	// Sensors - Waster Water Sump
	{attribute 'OPC.UA.DA' := '1'}
  	{attribute 'OPC.UA.DA.StructuredType' := '1'}
	fbSensor_WWS_LSLL : FB_Sensor_SICKLevelSwitch_GRF18S(SensorID:= 'SU3-LSLL' , SensorDescr:= 'Waste Water Sump Level Switch - LOW LOW', SensorType:= E_SensorType.Analogue);
	{attribute 'OPC.UA.DA' := '1'}
  	{attribute 'OPC.UA.DA.StructuredType' := '1'}
	fbSensor_WWS_LSL : FB_Sensor_SICKLevelSwitch_GRF18S(SensorID:= 'SU3-LSL' , SensorDescr:= 'Waste Water Sump Level Switch - LOW', SensorType:= E_SensorType.Analogue);
	{attribute 'OPC.UA.DA' := '1'}
  	{attribute 'OPC.UA.DA.StructuredType' := '1'}
	fbSensor_WWS_LSH : FB_Sensor_SICKLevelSwitch_GRF18S(SensorID:= 'SU3-LSH' , SensorDescr:= 'Waste Water Sump Level Switch - HIGH', SensorType:= E_SensorType.Analogue);
	
	
	// Sensors - Waster Water Tank
	{attribute 'OPC.UA.DA' := '1'}
  	{attribute 'OPC.UA.DA.StructuredType' := '1'}
	fbSensor_WWT_LIT1 : FB_Sensor_4_20mA_Generic(SensorID:= 'TK1-LIT1', SensorDescr:= 'Waste Water Tank Level Transmitter 1' , SensorType:= E_SensorType.Analogue);
	{attribute 'OPC.UA.DA' := '1'}
  	{attribute 'OPC.UA.DA.StructuredType' := '1'} 
	fbSensor_WWT_LIT2 : FB_Sensor_4_20mA_Generic(SensorID:= 'TK1-LIT1', SensorDescr:= 'Waste Water Tank Level Transmitter 2' , SensorType:= E_SensorType.Analogue);
	{attribute 'OPC.UA.DA' := '1'}
  	{attribute 'OPC.UA.DA.StructuredType' := '1'}
 	fbSensor_WWT_LIT : FB_DualRedundantSensor(SensorID:= 'TK1-LIT', SensorDescr:= 'Waste Water Tank Level', SensorType:= E_SensorType.Analogue);
	
	// Actuated Valves 
	{attribute 'OPC.UA.DA' := '1'}
  	{attribute 'OPC.UA.DA.StructuredType' := '1'}
	fbValve_TownWaterSupply: FB_Valve_ONOFF_woMonitoring(ValveID:= 'TK1-V2', ValveDescr:= 'Town Water Supply Valve');
	{attribute 'OPC.UA.DA' := '1'}
  	{attribute 'OPC.UA.DA.StructuredType' := '1'}
	fbValve_DosingSupply: FB_Valve_ONOFF_woMonitoring(ValveID:= 'PU1-V1', ValveDescr:= 'Dosing Circuit Supply Valve');
	{attribute 'OPC.UA.DA' := '1'}
  	{attribute 'OPC.UA.DA.StructuredType' := '1'}
	fbValve_DM1Supply: FB_Valve_ONOFF_woMonitoring(ValveID:= 'PU1-V2', ValveDescr:= 'Dosing Machine 1 Supply Valve' );
	{attribute 'OPC.UA.DA' := '1'}
  	{attribute 'OPC.UA.DA.StructuredType' := '1'} 
	fbValve_DM2Supply: FB_Valve_ONOFF_woMonitoring(ValveID:= 'PU1-V3', ValveDescr:= 'Dosing Machine 2 Supply Valve' );
	{attribute 'OPC.UA.DA' := '1'}
  	{attribute 'OPC.UA.DA.StructuredType' := '1'}
	fbValve_SeedStackSupply: FB_Valve_ONOFF_woMonitoring(ValveID:= 'PU1-V4', ValveDescr:= 'Seedling Stack Supply Valve' );
	{attribute 'OPC.UA.DA' := '1'}
  	{attribute 'OPC.UA.DA.StructuredType' := '1'}
	fbValve_SDRSoakSupply: FB_Valve_ONOFF_woMonitoring(ValveID:= 'PU1-V5', ValveDescr:= 'SDR Soak Supply Valve' );
	{attribute 'OPC.UA.DA' := '1'}
  	{attribute 'OPC.UA.DA.StructuredType' := '1'} 
	fbValve_WashSupply: FB_Valve_ONOFF_woMonitoring(ValveID:= 'PU1-V6', ValveDescr:= 'Pressure Wash Pumps Supply' );
	{attribute 'OPC.UA.DA' := '1'}
  	{attribute 'OPC.UA.DA.StructuredType' := '1'}
	fbValve_FogMistSupply: FB_Valve_ONOFF_woMonitoring(ValveID:= 'PU1-V7', ValveDescr:= 'Fog and Misting Pumps Supply' ); 

	// Tanks and Sumps
	{attribute 'OPC.UA.DA' := '1'}
  	{attribute 'OPC.UA.DA.StructuredType' := '1'}
	fbTank_CWTA: FB_Tank(TankID:= 'TK1A', TankDescr:= 'Clean Water Tank A');
	{attribute 'OPC.UA.DA' := '1'}
  	{attribute 'OPC.UA.DA.StructuredType' := '1'}
	fbTank_CWTB: FB_Tank(TankID:= 'TK1B', TankDescr:= 'Clean Water Tank B');
	{attribute 'OPC.UA.DA' := '1'}
  	{attribute 'OPC.UA.DA.StructuredType' := '1'}
	fbTank_WWT: FB_Tank(TankID:= 'TK2', TankDescr:= 'Waste Water Tank');
	{attribute 'OPC.UA.DA' := '1'}
  	{attribute 'OPC.UA.DA.StructuredType' := '1'}
	fbSump_WWS: FB_Tank(TankID:= 'TK3', TankDescr:= 'Waste Water Sump');
	
	
	// Control Loops
{attribute 'OPC.UA.DA' := '0'}
	fbControlLoop_Dosing: FB_ControlLoop_pH(
								DosingPump_phUp := fbDosingPump_phUp, 
								DosingPump_phDOwn := fbDosingPump_phDown, 
								Sensor_PH := fbSensor_PH, 
								Sensor_TEMP := fbSensor_TMP);
	
	
	// Package all components into structure to pass to sub-FBs 
	// This ST is populated by calling the populateComponents method
	{attribute 'OPC.UA.DA' := '0'} 
	stAllComponents: ST_WTRComponents;
	
	
	// Interlocks
	{attribute 'OPC.UA.DA' := '1'}
  	{attribute 'OPC.UA.DA.StructuredType' := '1'}
	fbInterlocks: FB_InterlockManager;
	
	{attribute 'OPC.UA.DA' := '1'}
	bInCalibration: BOOL := FALSE;
	
	// Sequence Manager & Sequences
	{attribute 'OPC.UA.DA' := '0'}
	fbSeqWTRMain: FB_SequenceWTR_Main;
	{attribute 'OPC.UA.DA' := '0'}
	fbSeqWTRMCalibrate: FB_SequenceWTR_Calibrate;
	{attribute 'OPC.UA.DA' := '0'}
	aSeqs: ARRAY[1..5] OF FB_SequenceBase;
	
END_VAR

IF GVL.bAutoUpdateDeviceState THEN
	simulation();       //  <<<----------------- FOR TESTING ONLY, delete this when not being used (it changes devices statet to the target state automatically)
END_IF

IF bIsFirstRun  THEN
	devices_init();	
	sequence_init();
	bIsFirstRun := FALSE;
END_IF


scanOPCInputs();
fbSequenceManager(aSequences := aSeqs, fbCurrentSequence := aSeqs[1]);
fbControlLoop_Dosing();

IF GVL.bEnableInterlocks_DM THEN
	interlocks();
END_IF

devices_update();

METHOD checkWaterQuality : BOOL
VAR_INPUT
END_VAR
(*

checkWaterQuality := TRUE;

IF fbSensor_PH.getValue() > stInputs.PH_HIGH_Limit OR 
	fbSensor_PH.getValue() < stInputs.PH_LOW_Limit THEN
	
	checkWaterQuality := FALSE;
	// Raise an event to alert that PH is out of range
END_IF

IF fbSensor_TMP.getValue() > stInputs.Temp_HIGH_Limit OR
	fbSensor_TMP.getValue() < stInputs.Temp_LOW_Limit THEN
	
	checkWaterQuality := FALSE;
	// Raise an event to alert that temp is out of range
END_IF

*)
END_METHOD

METHOD devices_init : BOOL
VAR
	VarInfo : __SYSTEM.VAR_INFO;
END_VAR
fbSump_WWS.fbSensor_LL := fbSensor_WWS_LSLL;
fbSump_WWS.fbSensor_L := fbSensor_WWS_LSL;
fbSump_WWS.fbSensor_H := fbSensor_WWS_LSH;
fbSump_WWS.fbSensor_HH := fbSensor_WWT_LIT;
fbSump_WWS.fbSensor_LIT := fbSensor_WWT_LIT;

fbTank_CWTA.fbSensor_LL := fbSensor_CWT_A_LSLL;
fbTank_CWTA.fbSensor_L := fbSensor_CWT_A_LSL;
fbTank_CWTA.fbSensor_H := fbSensor_CWT_A_LSH;
fbTank_CWTA.fbSensor_HH := fbSensor_CWT_A_LSHH;
fbTank_CWTA.fbSensor_LIT := fbSensor_CWT_A_LSHH;

fbTank_CWTB.fbSensor_LL := fbSensor_CWT_A_LSLL;
fbTank_CWTB.fbSensor_L := fbSensor_CWT_A_LSL;
fbTank_CWTB.fbSensor_H := fbSensor_CWT_A_LSH;
fbTank_CWTB.fbSensor_HH := fbSensor_CWT_A_LSHH;
fbTank_CWTB.fbSensor_LIT := fbSensor_CWT_A_LSHH;

fbTank_WWT.fbSensor_LL := fbSensor_CWT_A_LSLL;
fbTank_WWT.fbSensor_L := fbSensor_CWT_A_LSL;
fbTank_WWT.fbSensor_H := fbSensor_CWT_A_LSH;
fbTank_WWT.fbSensor_HH := fbSensor_CWT_A_LSHH;
fbTank_WWT.fbSensor_LIT := fbSensor_CWT_A_LSHH;




VarInfo := __VARINFO(fbDosingPump_phDown);
fbDosingPump_phDown.setVarID(VarID := VarInfo.Symbol);
VarInfo := __VARINFO(fbDosingPump_phUp);
fbDosingPump_phUp.setVarID(VarID := VarInfo.Symbol);
VarInfo := __VARINFO(fbDrumFilter_WasteWaterSump);
fbDrumFilter_WasteWaterSump.setVarID(VarID := VarInfo.Symbol);
VarInfo := __VARINFO(fbPump_CleanWaterPumpA);
fbPump_CleanWaterPumpA.setVarID(VarID := VarInfo.Symbol);
VarInfo := __VARINFO(fbPump_CleanWaterPumpB);
fbPump_CleanWaterPumpB.setVarID(VarID := VarInfo.Symbol);
VarInfo := __VARINFO(fbPump_WasteWaterSumpPumpA );
fbPump_WasteWaterSumpPumpA .setVarID(VarID := VarInfo.Symbol);
VarInfo := __VARINFO(fbPump_WasteWaterSumpPumpB );
fbPump_WasteWaterSumpPumpB .setVarID(VarID := VarInfo.Symbol);
VarInfo := __VARINFO(fbSensor_CWT_A_LIT );
fbSensor_CWT_A_LIT .setVarID(VarID := VarInfo.Symbol);
VarInfo := __VARINFO(fbSensor_CWT_A_LIT1 );
fbSensor_CWT_A_LIT1 .setVarID(VarID := VarInfo.Symbol);
VarInfo := __VARINFO(fbSensor_CWT_A_LIT2 );
fbSensor_CWT_A_LIT2 .setVarID(VarID := VarInfo.Symbol);
VarInfo := __VARINFO(fbSensor_CWT_A_LSH );
fbSensor_CWT_A_LSH .setVarID(VarID := VarInfo.Symbol);
VarInfo := __VARINFO(fbSensor_CWT_A_LSHH );
fbSensor_CWT_A_LSHH .setVarID(VarID := VarInfo.Symbol);
VarInfo := __VARINFO(fbSensor_CWT_A_LSL );
fbSensor_CWT_A_LSL .setVarID(VarID := VarInfo.Symbol);
VarInfo := __VARINFO(fbSensor_CWT_A_LSLL );
fbSensor_CWT_A_LSLL .setVarID(VarID := VarInfo.Symbol);
VarInfo := __VARINFO(fbSensor_CWT_B_LIT );
fbSensor_CWT_B_LIT .setVarID(VarID := VarInfo.Symbol);
VarInfo := __VARINFO(fbSensor_CWT_B_LIT1 );
fbSensor_CWT_B_LIT1 .setVarID(VarID := VarInfo.Symbol);
VarInfo := __VARINFO(fbSensor_CWT_B_LIT2 );
fbSensor_CWT_B_LIT2 .setVarID(VarID := VarInfo.Symbol);
VarInfo := __VARINFO(fbSensor_CWT_B_LSH );
fbSensor_CWT_B_LSH .setVarID(VarID := VarInfo.Symbol);
VarInfo := __VARINFO(fbSensor_CWT_B_LSHH );
fbSensor_CWT_B_LSHH .setVarID(VarID := VarInfo.Symbol);
VarInfo := __VARINFO(fbSensor_CWT_B_LSL );
fbSensor_CWT_B_LSL .setVarID(VarID := VarInfo.Symbol);
VarInfo := __VARINFO(fbSensor_CWT_B_LSLL );
fbSensor_CWT_B_LSLL .setVarID(VarID := VarInfo.Symbol);
VarInfo := __VARINFO(fbSensor_PH);
fbSensor_PH.setVarID(VarID := VarInfo.Symbol);
VarInfo := __VARINFO(fbSensor_PH1);
fbSensor_PH1.setVarID(VarID := VarInfo.Symbol);
VarInfo := __VARINFO(fbSensor_PH2);
fbSensor_PH2.setVarID(VarID := VarInfo.Symbol);
VarInfo := __VARINFO(fbSensor_TMP);
fbSensor_TMP.setVarID(VarID := VarInfo.Symbol);
VarInfo := __VARINFO(fbSensor_TMP1);
fbSensor_TMP1.setVarID(VarID := VarInfo.Symbol);
VarInfo := __VARINFO(fbSensor_TMP2);
fbSensor_TMP2.setVarID(VarID := VarInfo.Symbol);
VarInfo := __VARINFO(fbSensor_WWS_LSH );
fbSensor_WWS_LSH .setVarID(VarID := VarInfo.Symbol);
VarInfo := __VARINFO(fbSensor_WWS_LSL );
fbSensor_WWS_LSL .setVarID(VarID := VarInfo.Symbol);
VarInfo := __VARINFO(fbSensor_WWS_LSLL );
fbSensor_WWS_LSLL .setVarID(VarID := VarInfo.Symbol);
VarInfo := __VARINFO(fbSensor_WWT_LIT );
fbSensor_WWT_LIT .setVarID(VarID := VarInfo.Symbol);
VarInfo := __VARINFO(fbSensor_WWT_LIT1 );
fbSensor_WWT_LIT1 .setVarID(VarID := VarInfo.Symbol);
VarInfo := __VARINFO(fbSensor_WWT_LIT2 );
fbSensor_WWT_LIT2 .setVarID(VarID := VarInfo.Symbol);
VarInfo := __VARINFO(fbSump_WWS);
fbSump_WWS.setVarID(VarID := VarInfo.Symbol);
VarInfo := __VARINFO(fbTank_CWTA);
fbTank_CWTA.setVarID(VarID := VarInfo.Symbol);
VarInfo := __VARINFO(fbTank_CWTB);
fbTank_CWTB.setVarID(VarID := VarInfo.Symbol);
VarInfo := __VARINFO(fbTank_WWT);
fbTank_WWT.setVarID(VarID := VarInfo.Symbol);
VarInfo := __VARINFO(fbUnit_OzoneGenerator);
fbUnit_OzoneGenerator.setVarID(VarID := VarInfo.Symbol);
VarInfo := __VARINFO(fbUnit_RO_EDI);
fbUnit_RO_EDI.setVarID(VarID := VarInfo.Symbol);
VarInfo := __VARINFO(fbValve_DM1Supply);
fbValve_DM1Supply.setVarID(VarID := VarInfo.Symbol);
VarInfo := __VARINFO(fbValve_DM2Supply);
fbValve_DM2Supply.setVarID(VarID := VarInfo.Symbol);
VarInfo := __VARINFO(fbValve_DosingSupply);
fbValve_DosingSupply.setVarID(VarID := VarInfo.Symbol);
VarInfo := __VARINFO(fbValve_FogMistSupply);
fbValve_FogMistSupply.setVarID(VarID := VarInfo.Symbol);
VarInfo := __VARINFO(fbValve_SDRSoakSupply);
fbValve_SDRSoakSupply.setVarID(VarID := VarInfo.Symbol);
VarInfo := __VARINFO(fbValve_SeedStackSupply);
fbValve_SeedStackSupply.setVarID(VarID := VarInfo.Symbol);
VarInfo := __VARINFO(fbValve_TownWaterSupply);
fbValve_TownWaterSupply.setVarID(VarID := VarInfo.Symbol);
VarInfo := __VARINFO(fbValve_WashSupply);
fbValve_WashSupply.setVarID(VarID := VarInfo.Symbol);




stAllComponents.fbDosingPump_phUp :=  ADR( fbDosingPump_phUp);
stAllComponents.fbDosingPump_phDown :=  ADR( fbDosingPump_phDown);
stAllComponents.fbPump_CleanWaterPumpA :=  ADR( fbPump_CleanWaterPumpA);
stAllComponents.fbPump_CleanWaterPumpB :=  ADR( fbPump_CleanWaterPumpB);
stAllComponents.fbPump_WasteWaterSumpPumpA :=  ADR( fbPump_WasteWaterSumpPumpA);
stAllComponents.fbPump_WasteWaterSumpPumpB :=  ADR( fbPump_WasteWaterSumpPumpB);
stAllComponents.fbUnit_OzoneGenerator :=  ADR( fbUnit_OzoneGenerator);
stAllComponents.fbUnit_RO_EDI := ADR( fbUnit_RO_EDI);
stAllComponents.fbDrumFilter_WasteWaterSump :=  ADR( fbDrumFilter_WasteWaterSump);
stAllComponents.fbSensor_PH1 :=  ADR( fbSensor_PH1);
stAllComponents.fbSensor_PH2 :=  ADR( fbSensor_PH2);
stAllComponents.fbSensor_PH :=  ADR( fbSensor_PH);
stAllComponents.fbSensor_TMP1 :=  ADR( fbSensor_TMP1);
stAllComponents.fbSensor_TMP2 :=  ADR( fbSensor_TMP2);
stAllComponents.fbSensor_TMP :=  ADR( fbSensor_TMP);
stAllComponents.fbSensor_CWT_A_LIT1 :=  ADR( fbSensor_CWT_A_LIT1);
stAllComponents.fbSensor_CWT_A_LIT2 :=  ADR( fbSensor_CWT_A_LIT2);
stAllComponents.fbSensor_CWT_A_LIT :=  ADR( fbSensor_CWT_A_LIT);
stAllComponents.fbSensor_CWT_A_LSLL :=  ADR( fbSensor_CWT_A_LSLL);
stAllComponents.fbSensor_CWT_A_LSL :=  ADR( fbSensor_CWT_A_LSL);
stAllComponents.fbSensor_CWT_A_LSH :=  ADR( fbSensor_CWT_A_LSH);
stAllComponents.fbSensor_CWT_A_LSHH :=  ADR( fbSensor_CWT_A_LSHH);
stAllComponents.fbSensor_CWT_B_LIT1 :=  ADR( fbSensor_CWT_B_LIT1);
stAllComponents.fbSensor_CWT_B_LIT2 :=  ADR( fbSensor_CWT_B_LIT2);
stAllComponents.fbSensor_CWT_B_LIT :=  ADR( fbSensor_CWT_B_LIT);
stAllComponents.fbSensor_CWT_B_LSLL :=  ADR( fbSensor_CWT_B_LSLL);
stAllComponents.fbSensor_CWT_B_LSL :=  ADR( fbSensor_CWT_B_LSL);
stAllComponents.fbSensor_CWT_B_LSH :=  ADR( fbSensor_CWT_B_LSH);
stAllComponents.fbSensor_CWT_B_LSHH :=  ADR( fbSensor_CWT_B_LSHH);
stAllComponents.fbSensor_WWS_LSLL :=  ADR( fbSensor_WWS_LSLL);
stAllComponents.fbSensor_WWS_LSL :=  ADR( fbSensor_WWS_LSL);
stAllComponents.fbSensor_WWS_LSH :=  ADR( fbSensor_WWS_LSH);
stAllComponents.fbSensor_WWT_LIT1 :=  ADR( fbSensor_WWT_LIT1);
stAllComponents.fbSensor_WWT_LIT2 :=  ADR( fbSensor_WWT_LIT2);
stAllComponents.fbSensor_WWT_LIT :=  ADR( fbSensor_WWT_LIT);
stAllComponents.fbValve_TownWaterSupply :=  ADR( fbValve_TownWaterSupply);
stAllComponents.fbValve_DosingSupply :=  ADR( fbValve_DosingSupply);
stAllComponents.fbValve_DM1Supply :=  ADR( fbValve_DM1Supply);
stAllComponents.fbValve_DM2Supply :=  ADR( fbValve_DM2Supply);
stAllComponents.fbValve_SeedStackSupply :=  ADR( fbValve_SeedStackSupply);
stAllComponents.fbValve_SDRSoakSupply :=  ADR( fbValve_SDRSoakSupply);
stAllComponents.fbValve_WashSupply :=  ADR( fbValve_WashSupply);
stAllComponents.fbValve_FogMistSupply :=  ADR( fbValve_FogMistSupply);
stAllComponents.fbTank_CWTA :=  ADR( fbTank_CWTA);
stAllComponents.fbTank_CWTB :=  ADR( fbTank_CWTB);
stAllComponents.fbTank_WWT :=  ADR( fbTank_WWT);
stAllComponents.fbSump_WWS :=  ADR( fbSump_WWS);


aAllComponents[1]  :=  ADR(fbPump_CleanWaterPumpA );
aAllComponents[2]  :=  ADR(fbPump_CleanWaterPumpB );
aAllComponents[3]  :=  ADR(fbPump_WasteWaterSumpPumpA  );
aAllComponents[4]  :=  ADR(fbPump_WasteWaterSumpPumpB  );
aAllComponents[5]  :=  ADR(fbUnit_OzoneGenerator );
aAllComponents[6]  :=  ADR(fbDrumFilter_WasteWaterSump );
aAllComponents[7]  :=  ADR(fbUnit_RO_EDI );
aAllComponents[8]  :=  ADR(fbSensor_PH1 );
aAllComponents[9]  :=  ADR(fbSensor_PH2 );
aAllComponents[10]  :=  ADR(fbSensor_PH );
aAllComponents[11]  :=  ADR(fbSensor_TMP1 );
aAllComponents[12]  :=  ADR(fbSensor_TMP2 );
aAllComponents[13]  :=  ADR(fbSensor_TMP );
aAllComponents[14]  :=  ADR(fbSensor_CWT_A_LIT1  );
aAllComponents[15]  :=  ADR(fbSensor_CWT_A_LIT2  );
aAllComponents[16]  :=  ADR(fbSensor_CWT_A_LIT  );
aAllComponents[17]  :=  ADR(fbSensor_CWT_A_LSLL  );
aAllComponents[18]  :=  ADR(fbSensor_CWT_A_LSL  );
aAllComponents[19]  :=  ADR(fbSensor_CWT_A_LSH  );
aAllComponents[20]  :=  ADR(fbSensor_CWT_A_LSHH  );
aAllComponents[21]  :=  ADR(fbSensor_CWT_B_LIT1  );
aAllComponents[22]  :=  ADR(fbSensor_CWT_B_LIT2  );
aAllComponents[23]  :=  ADR(fbSensor_CWT_B_LIT  );
aAllComponents[24]  :=  ADR(fbSensor_CWT_B_LSLL  );
aAllComponents[25]  :=  ADR(fbSensor_CWT_B_LSL  );
aAllComponents[26]  :=  ADR(fbSensor_CWT_B_LSH  );
aAllComponents[27]  :=  ADR(fbSensor_CWT_B_LSHH  );
aAllComponents[28]  :=  ADR(fbSensor_WWS_LSLL  );
aAllComponents[29]  :=  ADR(fbSensor_WWS_LSL  );
aAllComponents[30]  :=  ADR(fbSensor_WWS_LSH  );
aAllComponents[31]  :=  ADR(fbSensor_WWT_LIT1  );
aAllComponents[32]  :=  ADR(fbSensor_WWT_LIT2  );
aAllComponents[33]  :=  ADR(fbSensor_WWT_LIT  );
aAllComponents[34]  :=  ADR(fbValve_TownWaterSupply );
aAllComponents[35]  :=  ADR(fbValve_DosingSupply );
aAllComponents[36]  :=  ADR(fbValve_DM1Supply );
aAllComponents[37]  :=  ADR(fbValve_DM2Supply );
aAllComponents[38]  :=  ADR(fbValve_SeedStackSupply );
aAllComponents[39]  :=  ADR(fbValve_SDRSoakSupply );
aAllComponents[40]  :=  ADR(fbValve_WashSupply );
aAllComponents[41]  :=  ADR(fbValve_FogMistSupply );
aAllComponents[42]  :=  ADR(fbTank_CWTA );
aAllComponents[43]  :=  ADR(fbTank_CWTB );
aAllComponents[44]  :=  ADR(fbTank_WWT );
aAllComponents[45]  :=  ADR(fbSump_WWS );

nQtyComponents := 45;
devices_disable_All();
END_METHOD

METHOD devices_update : BOOL
VAR_INPUT
END_VAR
fbModbusMaster();

fbDosingPump_phUp(fbModbusMaster := fbModbusMaster);
fbDosingPump_phDown(fbModbusMaster := fbModbusMaster);
fbPump_CleanWaterPumpA(fbModbusMaster := fbModbusMaster);	 
fbPump_CleanWaterPumpB(fbModbusMaster := fbModbusMaster); 
fbPump_WasteWaterSumpPumpA();
fbPump_WasteWaterSumpPumpB();
fbUnit_OzoneGenerator();
fbDrumFilter_WasteWaterSump();
fbSensor_PH1();
fbSensor_PH2();
fbSensor_PH();
fbSensor_TMP1();
fbSensor_TMP2();
fbSensor_TMP();
fbSensor_CWT_A_LIT1(); 
fbSensor_CWT_A_LIT2();
fbSensor_CWT_A_LIT();
fbSensor_CWT_A_LSLL();
fbSensor_CWT_A_LSL();
fbSensor_CWT_A_LSH();
fbSensor_CWT_A_LSHH();
fbSensor_CWT_B_LIT1(); 
fbSensor_CWT_B_LIT2();
fbSensor_CWT_B_LIT();
fbSensor_CWT_B_LSLL();
fbSensor_CWT_B_LSL();
fbSensor_CWT_B_LSH();
fbSensor_CWT_B_LSHH();
fbSensor_WWS_LSLL();
fbSensor_WWS_LSL();
fbSensor_WWS_LSH();
fbSensor_WWT_LIT1(); 
fbSensor_WWT_LIT2();
fbSensor_WWT_LIT();
fbValve_TownWaterSupply();
fbValve_DosingSupply();
fbValve_DM1Supply(); 
fbValve_DM2Supply();
fbValve_SeedStackSupply();
fbValve_SDRSoakSupply(); 
fbValve_WashSupply();
fbValve_FogMistSupply(); 
fbTank_CWTA();
fbTank_CWTB();		
fbTank_WWT();	
fbSump_WWS();
END_METHOD

METHOD FB_init : BOOL
VAR_INPUT
	bInitRetains : BOOL; // if TRUE, the retain variables are initialized (warm start / cold start)
	bInCopyCode : BOOL;  // if TRUE, the instance afterwards gets moved into the copy code (online change)


END_VAR
END_METHOD

METHOD interlocks : BOOL
VAR_INPUT
END_VAR


fbInterlocks.init();



// Dosing Pump - PH Up Interlocks

							
fbInterlocks.update(
							Description:= 'PH Down Dosing Pump - RUNNING',
							InterlockType:= E_InterlockType.RunInterlock, 
							Subject_Device:= ADR(fbDosingPump_phUp), 
							Subject_State:= E_DeviceState.IDLE, 
							Signal:= fbDosingPump_phDown.getState() = E_DeviceState.RUNNING, 
							HoldSequence:=	TRUE );
					
							
fbInterlocks.update(
							Description:= 'Dosing Line Pressure - OUT OF RANGE',		
							InterlockType:= E_InterlockType.StartPermissive, 
							Subject_Device:= ADR(fbDosingPump_phUp), 
							Subject_State:= E_DeviceState.IDLE, 
							Signal:= fbSensor_DosingPIT1.getState() = E_DeviceState.OUT_OF_RANGE, 
							HoldSequence:=	FALSE );	
							
// Dosing Pump - PH Down Interlocks


fbInterlocks.update(
							Description:= 'PH Up Dosing Pump - RUNNING',		
							InterlockType:= E_InterlockType.RunInterlock, 
							Subject_Device:= ADR(fbDosingPump_phDown), 
							Subject_State:= E_DeviceState.IDLE, 
							Signal:= fbDosingPump_phUp.getState() = E_DeviceState.RUNNING, 
							HoldSequence:=	TRUE );
							
fbInterlocks.update(
							Description:= 'Dosing Line Pressure - OUT OF RANGE',		
							InterlockType:= E_InterlockType.RunInterlock, 
							Subject_Device:= ADR(fbDosingPump_phDown), 
							Subject_State:= E_DeviceState.IDLE, 
							Signal:= fbSensor_DosingPIT1.getState() = E_DeviceState.OUT_OF_RANGE, 
							HoldSequence:=	FALSE );

							
// Clean Water Pump A - Interlocks	


fbInterlocks.update(
							Description:= 'Clean Water Pump B - RUNNING', 
							InterlockType:= E_InterlockType.RunInterlock, 
							Subject_Device:= ADR(fbPump_CleanWaterPumpA), 
							Subject_State:= E_DeviceState.IDLE, 
							Signal:= fbPump_CleanWaterPumpB.getState() = E_DeviceState.RUNNING, 
							HoldSequence:= TRUE);

fbInterlocks.update(
							Description:= 'Pressure Transmitter - OUT OF RANGE', 
							InterlockType:= E_InterlockType.RunInterlock, 
							Subject_Device:= ADR(fbPump_CleanWaterPumpA), 
							Subject_State:= E_DeviceState.IDLE, 
							Signal:= fbSensor_MainPumpPIT1.getState() = E_DeviceState.OUT_OF_RANGE, 
							HoldSequence:= TRUE);

fbInterlocks.update(
							Description:= 'Clean Water Tank (A) - LOW LOW Level', 
							InterlockType:= E_InterlockType.RunInterlock, 
							Subject_Device:= ADR(fbPump_CleanWaterPumpA), 
							Subject_State:= E_DeviceState.IDLE, 
							Signal:= fbTank_CWTA.getState() = E_DeviceState.LOW_LOW, 
							HoldSequence:= TRUE);

fbInterlocks.update(
							Description:= 'Clean Water Tank (B) - LOW LOW Level', 
							InterlockType:= E_InterlockType.RunInterlock, 
							Subject_Device:= ADR(fbPump_CleanWaterPumpA), 
							Subject_State:= E_DeviceState.IDLE, 
							Signal:= fbTank_CWTB.getState() = E_DeviceState.LOW_LOW, 
							HoldSequence:= TRUE);
							
fbInterlocks.update(
							Description:= 'Valve Combination - DM1, DM2, Recirc, Fog, SDR, Seedstack and Wash - CLOSED', 
							InterlockType:= E_InterlockType.RunInterlock, 
							Subject_Device:= ADR(fbPump_CleanWaterPumpA), 
							Subject_State:= E_DeviceState.IDLE, 
							Signal:= fbTank_CWTB.getState() = E_DeviceState.LOW_LOW, 
							HoldSequence:= TRUE);

// Clean Water Pump B - Interlocks	


fbInterlocks.update(
							Description:= 'Clean Water Pump A - RUNNING', 
							InterlockType:= E_InterlockType.RunInterlock, 
							Subject_Device:= ADR(fbPump_CleanWaterPumpB), 
							Subject_State:= E_DeviceState.IDLE, 
							Signal:= fbPump_CleanWaterPumpA.getState() = E_DeviceState.RUNNING, 
							HoldSequence:= TRUE);

fbInterlocks.update(
							Description:= 'Pressure Transmitter - OUT OF RANGE', 
							InterlockType:= E_InterlockType.RunInterlock, 
							Subject_Device:= ADR(fbPump_CleanWaterPumpB), 
							Subject_State:= E_DeviceState.IDLE, 
							Signal:= fbSensor_MainPumpPIT1.getState() = E_DeviceState.OUT_OF_RANGE, 
							HoldSequence:= TRUE);

fbInterlocks.update(
							Description:= 'Clean Water Tank (A) - LOW LOW Level', 
							InterlockType:= E_InterlockType.RunInterlock, 
							Subject_Device:= ADR(fbPump_CleanWaterPumpB), 
							Subject_State:= E_DeviceState.IDLE, 
							Signal:= fbTank_CWTA.getState() = E_DeviceState.LOW_LOW, 
							HoldSequence:= TRUE);

fbInterlocks.update(
							Description:= 'Clean Water Tank (B) - LOW LOW Level', 
							InterlockType:= E_InterlockType.RunInterlock, 
							Subject_Device:= ADR(fbPump_CleanWaterPumpB), 
							Subject_State:= E_DeviceState.IDLE, 
							Signal:= fbTank_CWTB.getState() = E_DeviceState.LOW_LOW, 
							HoldSequence:= TRUE);
							
fbInterlocks.update(
							Description:= 'Valve Combination - DM1, DM2, Recirc, Fog, SDR, Seedstack and Wash - CLOSED', 
							InterlockType:= E_InterlockType.RunInterlock, 
							Subject_Device:= ADR(fbPump_CleanWaterPumpB), 
							Subject_State:= E_DeviceState.IDLE, 
							Signal:= fbTank_CWTB.getState() = E_DeviceState.LOW_LOW, 
							HoldSequence:= TRUE);

// Waste Water Sump (WWS) Pump A							
							
fbInterlocks.update(
							Description:= 'Waste Water Sump Pump B - RUNNING', 
							InterlockType:= E_InterlockType.RunInterlock, 
							Subject_Device:= ADR(fbPump_WasteWaterSumpPumpA), 
							Subject_State:= E_DeviceState.IDLE, 
							Signal:= fbPump_WasteWaterSumpPumpB.getState() = E_DeviceState.RUNNING, 
							HoldSequence:= TRUE);
							
fbInterlocks.update(
							Description:= 'Waste Water Sump - LOW LOW Level', 
							InterlockType:= E_InterlockType.RunInterlock, 
							Subject_Device:= ADR(fbPump_WasteWaterSumpPumpA), 
							Subject_State:= E_DeviceState.IDLE, 
							Signal:= fbSump_WWS.getState() = E_DeviceState.LOW_LOW, 
							HoldSequence:= TRUE);		


// Waste Water Sump (WWS) Pump B							
							
fbInterlocks.update(
							Description:= 'Waste Water Sump Pump A - RUNNING', 
							InterlockType:= E_InterlockType.RunInterlock, 
							Subject_Device:= ADR(fbPump_WasteWaterSumpPumpB), 
							Subject_State:= E_DeviceState.IDLE, 
							Signal:= fbPump_WasteWaterSumpPumpA.getState() = E_DeviceState.RUNNING, 
							HoldSequence:= TRUE);
							
fbInterlocks.update(
							Description:= 'Waste Water Sump - LOW LOW Level', 
							InterlockType:= E_InterlockType.RunInterlock, 
							Subject_Device:= ADR(fbPump_WasteWaterSumpPumpB), 
							Subject_State:= E_DeviceState.IDLE, 
							Signal:= fbSump_WWS.getState() = E_DeviceState.LOW_LOW, 
							HoldSequence:= TRUE);		

// Ozone Generator (this is probably changint to a UV filter

fbInterlocks.update(
							Description:= 'Dosing line pressure - OUT OF RANGE', 
							InterlockType:= E_InterlockType.RunInterlock, 
							Subject_Device:= ADR(fbUnit_OzoneGenerator), 
							Subject_State:= E_DeviceState.OFF, 
							Signal:= fbSensor_DosingPIT1.getState() = E_DeviceState.OUT_OF_RANGE, 
							HoldSequence:= FALSE);			

fbInterlocks.update(
							Description:= 'Dosing line valve - CLOSED', 
							InterlockType:= E_InterlockType.RunInterlock, 
							Subject_Device:= ADR(fbUnit_OzoneGenerator), 
							Subject_State:= E_DeviceState.OFF, 
							Signal:= fbValve_DosingSupply.getState() = E_DeviceState.CLOSED, 
							HoldSequence:= FALSE);	

// RO / EDI SKid Interlocks

fbInterlocks.update(
							Description:= 'Waste Water Tank - LOW LOW Level', 
							InterlockType:= E_InterlockType.RunInterlock, 
							Subject_Device:= ADR(fbUnit_RO_EDI), 
							Subject_State:= E_DeviceState.OFF, 
							Signal:= fbTank_WWT.getState() = E_DeviceState.LOW_LOW, 
							HoldSequence:= TRUE);	
							
fbInterlocks.update(
							Description:= 'Clean Water Tank (A) - HIGH HIGH Level', 
							InterlockType:= E_InterlockType.RunInterlock, 
							Subject_Device:= ADR(fbUnit_RO_EDI), 
							Subject_State:= E_DeviceState.OFF, 
							Signal:= fbTank_CWTA.getState() = E_DeviceState.HIGH_HIGH, 
							HoldSequence:= TRUE);	
							
fbInterlocks.update(
							Description:= 'Clean Water Tank (B) - HIGH HIGH Level', 
							InterlockType:= E_InterlockType.RunInterlock, 
							Subject_Device:= ADR(fbUnit_RO_EDI), 
							Subject_State:= E_DeviceState.OFF, 
							Signal:= fbTank_CWTB.getState() = E_DeviceState.HIGH_HIGH, 
							HoldSequence:= TRUE);	

// Drum Filter 

fbInterlocks.update(
							Description:= 'Waste Water Sump - LOW LOW Level', 
							InterlockType:= E_InterlockType.RunInterlock, 
							Subject_Device:= ADR(fbDrumFilter_WasteWaterSump), 
							Subject_State:= E_DeviceState.OFF, 
							Signal:= fbSump_WWS.getState() = E_DeviceState.LOW_LOW, 
							HoldSequence:= FALSE);	

// DM1 Supply Valve

fbInterlocks.update(
							Description:= 'Water Quality (EC,pH,ORP,DO and temp) - OUT OF RANGE',
							InterlockType:= E_InterlockType.RunInterlock, 
							Subject_Device:= ADR(fbValve_DM1Supply), 
							Subject_State:= E_DeviceState.CLOSED, 
							Signal:= checkWaterQuality(), 
							HoldSequence:= FALSE);	


// DM2 Supply Valve							
							
fbInterlocks.update(
							Description:= 'Water Quality (EC,pH,ORP,DO and temp) - OUT OF RANGE',
							InterlockType:= E_InterlockType.RunInterlock, 
							Subject_Device:= ADR(fbValve_DM2Supply), 
							Subject_State:= E_DeviceState.CLOSED, 
							Signal:= checkWaterQuality(), 
							HoldSequence:= FALSE);							

							
// Dosing Recirc Supply
							
fbInterlocks.update(
							Description:= 'Water Quality Sensors Being Calibrated',
							InterlockType:= E_InterlockType.RunInterlock, 
							Subject_Device:= ADR(fbValve_DosingSupply), 
							Subject_State:= E_DeviceState.CLOSED, 
							Signal:= bInCalibration,
							HoldSequence:= FALSE);		

// Fog Misting Supply						
							
fbInterlocks.update(
							Description:= 'Water Quality (EC,pH,ORP,DO and temp) - OUT OF RANGE',
							InterlockType:= E_InterlockType.RunInterlock, 
							Subject_Device:= ADR(fbValve_FogMistSupply), 
							Subject_State:= E_DeviceState.CLOSED, 
							Signal:= checkWaterQuality(), 
							HoldSequence:= FALSE);							

// SDR Soak Supply						
							
fbInterlocks.update(
							Description:= 'Water Quality (EC,pH,ORP,DO and temp) - OUT OF RANGE',
							InterlockType:= E_InterlockType.RunInterlock, 
							Subject_Device:= ADR(fbValve_SDRSoakSupply), 
							Subject_State:= E_DeviceState.CLOSED, 
							Signal:= checkWaterQuality(), 
							HoldSequence:= FALSE);									
							
							
// Seed Stack Supply						
							
fbInterlocks.update(
							Description:= 'Water Quality (EC,pH,ORP,DO and temp) - OUT OF RANGE',
							InterlockType:= E_InterlockType.RunInterlock, 
							Subject_Device:= ADR(fbValve_SeedStackSupply), 
							Subject_State:= E_DeviceState.CLOSED, 
							Signal:= checkWaterQuality(), 
							HoldSequence:= FALSE);				
							
							
											
fbInterlocks.execute();
END_METHOD

METHOD scanOPCInputs : BOOL
VAR_INPUT
END_VAR
(*
(*
			SEQUENCE CONTROL
*)


IF stInputs.Sequence_Selected <> fbSequenceManager.getCurrentSeq_ID() THEN // Selected sequence has been changed
	fbSequenceManager.stopSequence();
	devices_disable_All();
	fbSequenceManager.selectSequence(stInputs.Sequence_Selected);
	devices_enable_CurrSeq();
	//fbSequenceManager.startSequence(); // Automatically start sequence on change of sequence selected - can change this if required
END_IF


IF stInputs.Sequence_Ack_Interlock THEN
	fbSequenceManager.acknowledgePause();
	stInputs.Sequence_Ack_Interlock := FALSE;
END_IF


CASE stInputs.Sequence_Command OF
	E_SequenceState.RUN:
		IF fbSequenceManager.getState() <> E_SequenceState.RUN THEN
			fbSequenceManager.startSequence();
		END_IF
	E_SequenceState.STOP:
		IF fbSequenceManager.getState() <> E_SequenceState.STOP THEN
			fbSequenceManager.stopSequence();
		END_IF
	E_SequenceState.HOLD:
		IF fbSequenceManager.getState() <> E_SequenceState.HOLD THEN
			fbSequenceManager.pauseSequence();
		END_IF
END_CASE


(*
			WATER QUALITY LIMITS
*)


nPH_Low_Limit := stInputs.PH_LOW_Limit;
nPH_High_Limit := stInputs.PH_HIGH_Limit;
nPH_SetPoint := stInputs.PH_SetPoint;

nTemp_Low_Limit := stInputs.Temp_LOW_Limit;
nTemp_Low_Limit := stInputs.Temp_LOW_Limit;
nTemp_SetPoint := stInputs.Temp_SetPoint;


(*
			PRESSURE LIMITS
*)

nPressureMin_Dosing := stInputs.Dosing_Pressure_LOW_Limit;
nPressureMax_Dosing := stInputs.Dosing_Pressure_HIGH_Limit;

(*
			PUMP SELECTION
*)

bPump_CleanWaterPumpSelection_A_1_B_0 := stInputs.Pump_CleanWaterPumpSelection_A_1_B_0;
bPump_WasteWaterSumpPumpSelection_A_1_B_0 := stInputs.Pump_WasteWaterSumpPumpSelection_A_1_B_0;

(*
			ACTUATORS - PUMPS
*)

// Clean Water Pump A
fbPump_CleanWaterPumpA.setMode(Mode := stInputs.Pump_CleanWaterPumpA_Mode);
IF fbPump_CleanWaterPumpA.inManual() THEN
	fbPump_CleanWaterPumpA.setCommand(StateTarget := stInputs.Pump_CleanWaterPumpA_Command);
	fbPump_CleanWaterPumpA.setReference(RefSetPoint := stInputs.Pump_CleanWaterPumpA_CommandFrequency);
END_IF

// Clean Water Pump B
fbPump_CleanWaterPumpB.setMode(Mode := stInputs.Pump_CleanWaterPumpB_Mode);
IF fbPump_CleanWaterPumpB.inManual() THEN
	fbPump_CleanWaterPumpB.setCommand(StateTarget := stInputs.Pump_CleanWaterPumpB_Command);
	fbPump_CleanWaterPumpB.setReference(RefSetPoint := stInputs.Pump_CleanWaterPumpB_CommandFrequency);
END_IF


// Dosing Pump - PH UP
fbDosingPump_phUp.setMode(Mode := stInputs.DosingPump_phUp_Mode);
IF fbDosingPump_phUp.inManual() THEN
	fbDosingPump_phUp.setCommand(StateTarget := stInputs.DosingPump_phUp_Command);
	fbDosingPump_phUp.setDoseParams(DoseQtyMls:= stInputs.DosingPump_phUp_DoseQty_mls,
								DoseRateMlph:= stInputs.DosingPump_phUp_DoseRate_mlph);
END_IF
						
IF stInputs.DosingPump_phUp_ResetPumpStatistics THEN
	fbDosingPump_phUp.resetStatistics();
	stInputs.DosingPump_phUp_ResetPumpStatistics := FALSE;
END_IF

// Dosing Pump - PH Down
fbDosingPump_phDown.setMode(Mode := stInputs.DosingPump_phDown_Mode);
IF fbDosingPump_phDown.inManual() THEN
	fbDosingPump_phDown.setCommand(StateTarget := stInputs.DosingPump_phDown_Command);
	fbDosingPump_phDown.setDoseParams(DoseQtyMls:= stInputs.DosingPump_phDown_DoseQty_mls,
								DoseRateMlph:= stInputs.DosingPump_phDown_DoseRate_mlph);
END_IF
						
IF stInputs.DosingPump_phDown_ResetPumpStatistics THEN
	fbDosingPump_phDown.resetStatistics();
	stInputs.DosingPump_phDown_ResetPumpStatistics := FALSE;
END_IF

// Waste Water Sump (WWS) Pump A
fbPump_WasteWaterSumpPumpA.setMode(Mode := stInputs.Pump_WasteWaterSumpPumpA_Mode);
IF fbPump_WasteWaterSumpPumpA.inManual() THEN
	fbPump_WasteWaterSumpPumpA.setCommand(StateTarget := stInputs.Pump_WasteWaterSumpPumpA_Command);
END_IF

// Waste Water Sump (WWS) Pump B
fbPump_WasteWaterSumpPumpB.setMode(Mode := stInputs.Pump_WasteWaterSumpPumpB_Mode);
IF fbPump_WasteWaterSumpPumpB.inManual() THEN
	fbPump_WasteWaterSumpPumpB.setCommand(StateTarget := stInputs.Pump_WasteWaterSumpPumpB_Command);
END_IF


// Ozone Generator
fbUnit_OzoneGenerator.setMode(Mode := stInputs.Unit_OzoneGenerator_Mode);
IF fbUnit_OzoneGenerator.inManual() THEN
	fbUnit_OzoneGenerator.setCommand(StateTarget := stInputs.Unit_OzoneGenerator_Command);
END_IF

// Waste Water Sump Drum Filter
fbDrumFilter_WasteWaterSump.setMode(Mode := stInputs.DrumFilter_WasteWaterSump_Mode);
IF fbDrumFilter_WasteWaterSump.inManual() THEN
	fbDrumFilter_WasteWaterSump.setCommand(StateTarget := stInputs.DrumFilter_WasteWaterSump_Command);
END_IF

// RO/EDI Skid
fbUnit_RO_EDI.setMode(Mode := stInputs.Unit_RO_EDI_Mode);
IF fbUnit_RO_EDI.inManual() THEN
	fbUnit_RO_EDI.setCommand(StateTarget := stInputs.Unit_RO_EDI_Command);
END_IF




(*
			ACTUATORS - VALVES
*)

fbValve_DosingSupply.setMode(Mode := stInputs.Valve_DosingSupply_Mode);
IF fbValve_DosingSupply.inManual() THEN
	fbValve_DosingSupply.setCommand(StateTarget := stInputs.Valve_DosingSupply_Command);
END_IF

fbValve_DM1Supply.setMode(Mode := stInputs.Valve_DM1_Supply_Mode);
IF fbValve_DM1Supply.inManual() THEN
	fbValve_DM1Supply.setCommand(StateTarget := stInputs.Valve_DM1_Supply_Command);
END_IF

fbValve_DM2Supply.setMode(Mode := stInputs.Valve_DM2_Supply_Mode);
IF fbValve_DM2Supply.inManual() THEN
	fbValve_DM2Supply.setCommand(StateTarget := stInputs.Valve_DM2_Supply_Command);
END_IF

fbValve_DM2Supply.setMode(Mode := stInputs.Valve_DM2_Supply_Mode);
IF fbValve_DM2Supply.inManual() THEN
	fbValve_DM2Supply.setCommand(StateTarget := stInputs.Valve_DM2_Supply_Command);
END_IF

fbValve_SeedStackSupply.setMode(Mode := stInputs.Valve_Seedling_Stack_Mode);
IF fbValve_SeedStackSupply.inManual() THEN
	fbValve_SeedStackSupply.setCommand(StateTarget := stInputs.Valve_Seedling_Stack_Command);
END_IF

fbValve_SDRSoakSupply.setMode(Mode := stInputs.Valve_SDR_Machine_Soak_Mode);
IF fbValve_SDRSoakSupply.inManual() THEN
	fbValve_SDRSoakSupply.setCommand(StateTarget := stInputs.Valve_SDR_Machine_Soak_Command);
END_IF

fbValve_WashSupply.setMode(Mode := stInputs.Valve_Tray_Cleaning_Mode);
IF fbValve_WashSupply.inManual() THEN
	fbValve_WashSupply.setCommand(StateTarget := stInputs.Valve_Tray_Cleaning_Command);
END_IF

fbValve_FogMistSupply.setMode(Mode := stInputs.Valve_FogMisting_Mode);
IF fbValve_FogMistSupply.inManual() THEN
	fbValve_FogMistSupply.setCommand(StateTarget := stInputs.Valve_FogMisting_Command);
END_IF

fbValve_TownWaterSupply.setMode(Mode := stInputs.Valve_TownWater_Mode);
IF fbValve_TownWaterSupply.inManual() THEN
	fbValve_TownWaterSupply.setCommand(StateTarget := stInputs.Valve_TownWater_Command);
END_IF



fbControlLoop_Dosing.setParams(
								PHMaxDoseRate:= stInputs.ControlLoop_Dosing_PIDPH_MaxDoseRate, 
								PHMinDoseRate:= stInputs.ControlLoop_Dosing_PIDPH_MinDoseRate, 
								PHTimeBetweenDoses:= UINT_TO_TIME(stInputs.ControlLoop_Dosing_PIDPH_TimeBetweenDoses), 
								PHSetpoint:= stInputs.ControlLoop_Dosing_nPIDPHSetpoint , 
								PHSetpointBand:= stInputs.ControlLoop_Dosing_PIDPHSetpointBand, 
								PHManSyncVal:= stInputs.ControlLoop_Dosing_PIDPHManSyncVal, 
								PHSync:= stInputs.ControlLoop_Dosing_PIDPHSync, 
								PHHold:= stInputs.ControlLoop_Dosing_PIDPHHold, 
								PHMode:= stInputs.ControlLoop_Dosing_PIDPHMode, 
								PHCtrlCycleTime:= UINT_TO_TIME(stInputs.ControlLoop_Dosing_PIDPHCtrlCycleTime), 
								PHTaskCycleTime:= UINT_TO_TIME(stInputs.ControlLoop_Dosing_PIDPHTaskCycleTime), 
								PHKp:= stInputs.ControlLoop_Dosing_PIDPHKp, 
								PHTn:= UINT_TO_TIME(stInputs.ControlLoop_Dosing_PIDPHTn), 
								PHTv:= UINT_TO_TIME(stInputs.ControlLoop_Dosing_PIDPHTv), 
								PHTd:= UINT_TO_TIME(stInputs.ControlLoop_Dosing_PIDPHTd), 
								PHOutMaxLimit:= stInputs.ControlLoop_Dosing_PIDPHOutMaxLimit, 
								PHOutMinLimit:= stInputs.ControlLoop_Dosing_PIDPHOutMinLimit, 
								PHPInTheFeedbackPath:= stInputs.ControlLoop_Dosing_PIDPHPInTheFeedbackPath, 
								PHDInTheFeedbackPath:= stInputs.ControlLoop_Dosing_PIDPHDInTheFeedbackPath, 
								PHARWOnIPartOnly:= stInputs.ControlLoop_Dosing_PIDPHARWOnIPartOnly);



*)
END_METHOD

METHOD sequence_init : BOOL
VAR_INPUT
END_VAR
	fbSeqWTRMain(devices := stAllComponents);
	fbSeqWTRMain.populateSteps();
	
	fbSeqWTRMCalibrate(devices := stAllComponents);
	fbSeqWTRMCalibrate.populateSteps();

	aSeqs[1] := fbSeqWTRMain;
	aSeqs[2] := fbSeqWTRMCalibrate;
END_METHOD

METHOD simulation : BOOL
VAR_INPUT
END_VAR

fbDosingPump_phUp.runSimulation();
fbDosingPump_phDown.runSimulation();
fbPump_CleanWaterPumpA.runSimulation();	 
fbPump_CleanWaterPumpB.runSimulation();	 
fbPump_WasteWaterSumpPumpA.runSimulation();
fbPump_WasteWaterSumpPumpB.runSimulation();
fbUnit_OzoneGenerator.runSimulation();
fbDrumFilter_WasteWaterSump.runSimulation();

fbValve_TownWaterSupply.runSimulation();
fbValve_DosingSupply.runSimulation();
fbValve_DM1Supply.runSimulation(); 
fbValve_DM2Supply.runSimulation();
fbValve_SeedStackSupply.runSimulation();
fbValve_SDRSoakSupply.runSimulation(); 
fbValve_WashSupply.runSimulation();
fbValve_FogMistSupply.runSimulation();
END_METHOD

END_FUNCTION_BLOCK

// ---- POUs/06 Machines/Others/FB_Machine_WaterTreatment_RND.TcPOU
{attribute 'OPC.UA.DA.StructuredType' := '1'}
FUNCTION_BLOCK FB_Machine_WaterTreatment_RND EXTENDS FB_BaseMachine IMPLEMENTS I_Machine

VAR_IN_OUT

	{attribute 'OPC.UA.DA' := '0'} 
	stInputs: ST_INPUTS_WaterTreatment_RND;
END_VAR


VAR
	

	bIsFirstRun: BOOL := TRUE;

	
	// Tanks and Sumps
	{attribute 'OPC.UA.DA' := '1'}
  	{attribute 'OPC.UA.DA.StructuredType' := '1'}
	fbTank_CWTA: FB_Tank(TankID:= 'TK1', TankDescr:= 'Clean Water Tank');

	
	{attribute 'OPC.UA.DA' := '1'}
  	{attribute 'OPC.UA.DA.StructuredType' := '1'}
	fbSensor_CWT_A_LSH : FB_Sensor_SICKLevelSwitch_GRF18S(SensorID:= 'TK2A-LSH' , SensorDescr:= 'Clean Water Tank A Level Switch - HIGH', SensorType:= E_SensorType.Analogue);
	
	{attribute 'OPC.UA.DA' := '1'}
  	{attribute 'OPC.UA.DA.StructuredType' := '1'}
	fbUnit_RO_EDI: FB_Unit_RO_RND(UnitID:= 'U1', UnitDescr:= 'Reverse Osmosis (RO) & Electro De-Ionisation (EDI) Unit');
	
	
	// Package all components into structure to pass to sub-FBs 
	// This ST is populated by calling the populateComponents method
	{attribute 'OPC.UA.DA' := '0'} 
	stAllComponents: ST_RNDWTRComponents;
	
	// Interlocks
	{attribute 'OPC.UA.DA' := '1'}
  	{attribute 'OPC.UA.DA.StructuredType' := '1'}
	fbInterlocks: FB_InterlockManager;
	
	
	// Sequence Manager & Sequences
	{attribute 'OPC.UA.DA' := '0'}
	fbSeqWTRMain: FB_SequenceRNDWTR_Main;

	{attribute 'OPC.UA.DA' := '0'}
	aSeqs: ARRAY[1..5] OF FB_SequenceBase;
	
	fbTONStartSequence: TON := (PT := T#10s);
	
END_VAR

fbTONStartSequence();

IF GVL.bAutoUpdateDeviceState THEN
	simulation();       //  <<<----------------- FOR TESTING ONLY, delete this when not being used (it changes devices statet to the target state automatically)
END_IF

IF bIsFirstRun  THEN
	devices_init();	
	sequence_init();
	bIsFirstRun := FALSE;
	fbTONStartSequence(IN := TRUE);
END_IF

IF fbTONStartSequence.Q THEN
	fbSequenceManager.startSequence();
END_IF

scanOPCInputs();
fbSequenceManager(aSequences := aSeqs); //, fbCurrentSequence := aSeqs[1]);
interlocks();


IF GVL.bEnableInterlocks_DM THEN
	interlocks();
END_IF

devices_update();

METHOD checkWaterQuality : BOOL
VAR_INPUT
END_VAR
(*

checkWaterQuality := TRUE;

IF fbSensor_PH.getValue() > stInputs.PH_HIGH_Limit OR 
	fbSensor_PH.getValue() < stInputs.PH_LOW_Limit THEN
	
	checkWaterQuality := FALSE;
	// Raise an event to alert that PH is out of range
END_IF

IF fbSensor_TMP.getValue() > stInputs.Temp_HIGH_Limit OR
	fbSensor_TMP.getValue() < stInputs.Temp_LOW_Limit THEN
	
	checkWaterQuality := FALSE;
	// Raise an event to alert that temp is out of range
END_IF

*)
END_METHOD

METHOD devices_init : BOOL
VAR
	VarInfo : __SYSTEM.VAR_INFO;
END_VAR

fbTank_CWTA.fbSensor_H := fbSensor_CWT_A_LSH;



VarInfo := __VARINFO(fbSensor_CWT_A_LSH );
fbSensor_CWT_A_LSH .setVarID(VarID := VarInfo.Symbol);


VarInfo := __VARINFO(fbUnit_RO_EDI);
fbUnit_RO_EDI.setVarID(VarID := VarInfo.Symbol);



stAllComponents.fbUnit_RO_EDI := ADR( fbUnit_RO_EDI);
// stAllComponents.fbTank_CWTA :=  ADR( fbTank_CWTA);




aAllComponents[1]  :=  ADR(fbUnit_RO_EDI);
//aAllComponents[2]  :=  ADR(fbSensor_CWT_A_LSH );



nQtyComponents := 1;

devices_disable_All();
END_METHOD

METHOD devices_update : BOOL
VAR_INPUT
END_VAR


fbSensor_CWT_A_LSH();
//fbTank_CWTA();
fbUnit_RO_EDI();
END_METHOD

METHOD FB_init : BOOL
VAR_INPUT
	bInitRetains : BOOL; // if TRUE, the retain variables are initialized (warm start / cold start)
	bInCopyCode : BOOL;  // if TRUE, the instance afterwards gets moved into the copy code (online change)


END_VAR
END_METHOD

METHOD interlocks : BOOL
VAR_INPUT
END_VAR
fbInterlocks.init();

fbInterlocks.update(
							Description:= 'RND Clean Water Tank Is Full', 
							InterlockType:= E_InterlockType.RunInterlock, 
							Subject_Device:= ADR(fbUnit_RO_EDI), 
							Subject_State:= E_DeviceState.OFF, 
							Signal:= fbSensor_CWT_A_LSH.getValue() = 0, 
							HoldSequence:= FALSE);
							
fbInterlocks.execute();
END_METHOD

METHOD scanOPCInputs : BOOL
VAR_INPUT
END_VAR

(*
			SEQUENCE CONTROL
*)


IF stInputs.stSequenceManager.Sequence_Ack_Interlock THEN
	fbSequenceManager.acknowledgePause();
	stInputs.stSequenceManager.Sequence_Ack_Interlock := FALSE;
END_IF


CASE stInputs.stSequenceManager.Sequence_Command OF
	E_SequenceState.RUN:
		IF fbSequenceManager.getState() <> E_SequenceState.RUN THEN
			fbSequenceManager.startSequence();
			stInputs.stSequenceManager.Sequence_Command := E_SequenceState.WAIT;
		END_IF
	E_SequenceState.STOP:
		IF fbSequenceManager.getState() <> E_SequenceState.STOP THEN
			fbSequenceManager.stopSequence();
			stInputs.stSequenceManager.Sequence_Command := E_SequenceState.WAIT;
		END_IF
	E_SequenceState.HOLD:
		IF fbSequenceManager.getState() <> E_SequenceState.HOLD THEN
			fbSequenceManager.pauseSequence();
			stInputs.stSequenceManager.Sequence_Command := E_SequenceState.WAIT;
		END_IF
END_CASE
END_METHOD

METHOD sequence_init : BOOL
VAR_INPUT
END_VAR


fbSeqWTRMain(devices := stAllComponents);
fbSeqWTRMain.populateSteps();


aSeqs[1] := fbSeqWTRMain;
END_METHOD

METHOD simulation : BOOL
VAR_INPUT
END_VAR


//fbPump_CleanWaterPumpA.runSimulation();	 
//fbValve_TownWaterSupply.runSimulation();
//fbValve_DM1Supply.runSimulation(); 
//fbUnit_RO_EDI.runSimulation();
END_METHOD

END_FUNCTION_BLOCK

// ---- POUs/06 Machines/Others/FB_Stack_Controller.TcPOU
FUNCTION_BLOCK FB_Stack_Controller EXTENDS FB_BaseDevice
VAR_INPUT CONSTANT
	nLevels : INT;
	nStack : INT;
	nMaxStackEnvironmentZones: INT;
	nEnvironmentSensorModbusAddresses: ARRAY[0..2] OF ARRAY[0..10] OF UINT;
	nMaxLevelsPerStack: INT;
	sEnvironmentZoneNames: ARRAY[0..2] OF STRING;
END_VAR

VAR_IN_OUT
	fbModbus : FB_ModbusMaster;
END_VAR

VAR
	i : INT;
	//fbEnvironmentSensors : FB_SensorVirtual_Vaisala;
	fbEnvironmentZones 		: ARRAY[0..10] OF FB_SensorVirtual_Vaisala; 				// ARRAY[0..10] OF FB_SensorVirtual_Vaisala;
	fbLevelWaterControls 	: ARRAY[1..10] OF FB_LevelWaterControl; 	// ARRAY[1..nMaxLevelsPerStack] OF FB_LevelWaterControl;
	fbHumidityControl 		: FB_BangBangControl;
	fbCO2Control 			: FB_BangBangControl;
	fbTemperatureControl 	: FB_BangBangControl;
	
	{attribute 'OPC.UA.DA' := '1'}
	rStackHumidity : REAL;
	{attribute 'OPC.UA.DA' := '1'}
	rStackCO2 : REAL;
	{attribute 'OPC.UA.DA' := '1'}
	rStackTemp : REAL;
END_VAR



//fbEnvironmentSensors(nModbusUnitIDs := GVL.EnvironmentSensorModbusAddress, rMaxDiscrepency := 0.1, fbModbus := fbModbus);

// environment sensors for the stack zones
rStackHumidity := 0;
rStackCO2 := 0;
rStackTemp := 0;

FOR i := 0 TO nMaxStackEnvironmentZones DO
	fbEnvironmentZones[i](nModbusUnitIDs := nEnvironmentSensorModbusAddresses[i], rMaxDiscrepency := 0.1, fbModbus := fbModbus, sZoneName := sEnvironmentZoneNames[i]);
	rStackCO2 := rStackCO2 + fbEnvironmentZones[i].rCO2;
	rStackHumidity := rStackHumidity + fbEnvironmentZones[i].rHumidity;
	rStackTemp := rStackTemp + fbEnvironmentZones[i].rTemperature;
END_FOR

// calculate the average CO2 and humidity across the stack
rStackCO2 := rStackCO2 / (nMaxStackEnvironmentZones+1);
rStackHumidity := rStackHumidity / (nMaxStackEnvironmentZones+1);
rStackTemp := rStackTemp / (nMaxStackEnvironmentZones+1);

// control for humidity
fbHumidityControl(rCurrentValue := rStackHumidity, sParameterName := 'Humidity');
// bang bang control for CO2
fbCO2Control(rCurrentValue := rStackCO2, sParameterName := 'CO2');
// bang bang control for temperature
fbTemperatureControl(rCurrentValue := rStackTemp, sParameterName := 'Temperature');

// Function blocks which have an instance for every level...
FOR i := 1 TO nLevels DO
	// Irrigation valve
	fbLevelWaterControls[i](nLevel := i);
END_FOR

checkCropJobs();

METHOD checkCropJobs : BOOL
VAR_INPUT
END_VAR

// reset all crop jobs to false. Any active ones will be changed to true.
FOR i := 1 TO GVL.maxLevelsPerStack DO
	fbLevelWaterControls[i].bActiveCropJob := FALSE;
END_FOR

FOR i := 0 TO GVL.MaxCropJob DO
	// check if this crop job is coming FROM this stack
	IF Inputs.CropJobs[i].crop.stack = nStack AND Inputs.CropJobs[i].job_status > E_Job_Status.waiting AND Inputs.CropJobs[i].job_status < E_Job_Status.finished THEN
		fbLevelWaterControls[Inputs.CropJobs[i].crop.level].bActiveCropJob := TRUE;
	END_IF
	
	// check if this crop job is going TO this stack
	IF Inputs.CropJobs[i].stack = nStack AND Inputs.CropJobs[i].job_status > E_Job_Status.waiting AND Inputs.CropJobs[i].job_status < E_Job_Status.finished THEN
		fbLevelWaterControls[Inputs.CropJobs[i].level].bActiveCropJob := TRUE;
	END_IF

END_FOR
END_METHOD

METHOD FB_init : BOOL
VAR_INPUT
	bInitRetains : BOOL; // if TRUE, the retain variables are initialized (warm start / cold start)
	bInCopyCode : BOOL;  // if TRUE, the instance afterwards gets moved into the copy code (online change)
	
	ID : STRING;
	Description : STRING;
END_VAR

sID := ID;
sDescr := Description;
END_METHOD

END_FUNCTION_BLOCK

// ---- POUs/99 Utilities/FB_SensorVirtual_Vaisala.TcPOU
(*
	Manages a number of Vaisala sensor and reports the average values.
*)
{attribute 'OPC.UA.DA.StructuredType' := '1'}
FUNCTION_BLOCK FB_SensorVirtual_Vaisala EXTENDS FB_BaseDevice
VAR_INPUT
	nModbusUnitIDs: ARRAY[0..10] OF UINT;
	{attribute 'OPC.UA.DA' := '1'}
	rMaxDiscrepency : REAL;
	{attribute 'OPC.UA.DA' := '1'}
	sZoneName : STRING;
END_VAR

VAR_OUTPUT
	{attribute 'OPC.UA.DA' := '1'}
	rCO2 : REAL;
	{attribute 'OPC.UA.DA' := '1'}
	rTemperature : REAL;
	{attribute 'OPC.UA.DA' := '1'}
	rHumidity : REAL;
	{attribute 'OPC.UA.DA' := '1'}
	sError : STRING;
END_VAR

VAR
	fbSensors : ARRAY[0..10] OF FB_Sensor_VaisalaGMW90_R2_1; // FB_Sensor_VaisalaGMW90_R2;
	i : INT;
	rCO2_sum : REAL;
	rHum_sum : REAL;
	rTemp_sum : REAL;
	rCO2_min : REAL;
	rHum_min : REAL;
	rTemp_min : REAL;
	rCO2_max : REAL;
	rHum_max : REAL;
	rTemp_max : REAL;
	nSensorCount : INT;
	rRand : DRAND;
END_VAR

VAR_IN_OUT
	fbModbusManager : FB_ModbusManager;
END_VAR

rCO2_sum := 0;
rHum_sum := 0;
rTemp_sum := 0;
rCO2_min := 10000;
rHum_min := 10000;
rTemp_min := 10000;
rCO2_max := 0;
rHum_max := 0;
rTemp_max := 0;
nSensorCount := 0;

FOR i := 0 TO 10 DO
	
	IF nModbusUnitIDs[i] <> 0 THEN
		
		nSensorCount := nSensorCount + 1;
		
		fbSensors[i](nModbusUnitID := nModbusUnitIDs[i], fbModbusManager := fbModbusManager);		
		
		rCO2_sum := rCO2_sum + fbSensors[i].rCO2;
		rHum_sum := rHum_sum + fbSensors[i].rHumidity;
		rTemp_sum := rTemp_sum + fbSensors[i].rTemperature;
		
		rCO2_min := MIN(rCO2_min, fbSensors[i].rCO2);
		rHum_min := MIN(rHum_min, fbSensors[i].rHumidity);
		rTemp_min := MIN(rTemp_min, fbSensors[i].rTemperature);
		
		rCO2_max := MAX(rCO2_max, fbSensors[i].rCO2);
		rHum_max := MAX(rHum_max, fbSensors[i].rHumidity);
		rTemp_max := MAX(rTemp_max, fbSensors[i].rTemperature);
	
	END_IF

END_FOR

// calculate averages
IF nSensorCount <> 0 AND NOT GVL.bSimulateSensors THEN
	rCO2 := rCO2_sum / nSensorCount;
	rHumidity := rHum_sum / nSensorCount;
	rTemperature := rTemp_sum / nSensorCount;
END_IF

IF GVL.bSimulateSensors THEN
	rRand(Seed := 1);
	IF rCO2 < 10 THEN
		rCO2 := 250;
	END_IF
	IF rRand.Num > 0.999 THEN
		rCO2 := rCO2 * 1.01;
	ELSIF rRand.Num < 0.001 THEN
		rCO2 := rCO2 * 0.99;
	END_IF
	IF rHumidity < 10 THEN
		rHumidity := 60;
	END_IF
	IF rRand.Num > 0.999 THEN
		rHumidity := rHumidity * 1.01;
	ELSIF rRand.Num < 0.001 THEN
		rHumidity := rHumidity * 0.99;
	END_IF
	IF rTemperature < 5 THEN
		rTemperature := 18;
	END_IF
	IF rRand.Num > 0.999 THEN
		rTemperature := rTemperature * 1.01;
	ELSIF rRand.Num < 0.001 THEN
		rTemperature := rTemperature * 0.99;
	END_IF
END_IF

// Check sensor discrepencies
IF rCO2_min > 0 AND rHum_min > 0 AND rTemp_min > 0 THEN
	IF (ABS(rCO2_max - rCO2_min) / rCO2_min > rMaxDiscrepency) THEN
		sError := 'CO2 sensor discrepency';
	ELSIF (ABS(rHum_max - rHum_min) / rHum_min > rMaxDiscrepency) THEN
		sError := 'Humidity sensor discrepency';
	ELSIF (ABS(rTemp_max - rTemp_min) / rTemp_min > rMaxDiscrepency) THEN
		sError := 'Temperature sensor discrepency';
	ELSE
		sError := '';
	END_IF
ELSE
	sError := '';
END_IF

END_FUNCTION_BLOCK

// ---- POUs/06 Machines/Others/FB_Stack_Controller_RND.TcPOU
FUNCTION_BLOCK FB_Stack_Controller_RND EXTENDS FB_BaseDevice
VAR_INPUT CONSTANT
	 nLevels : INT;
	 nStack : INT;
END_VAR

VAR_IN_OUT
	fbModbusManager : FB_ModbusManager;
	fbHVAC: FB_System_RND_HVAC;
	stInputs: ST_INPUTS_RND_StackControl;
	stInputsHVAC: ST_HVAC;
END_VAR

VAR
	
	bFirstRun: BOOL := TRUE;
	i : INT;
	//fbEnvironmentSensors : FB_SensorVirtual_Vaisala;\
	nSensorModbusID_1: 		UINT;
	nSensorModbusID_2: 		UINT;
	sZoneName: 				STRING;
	
	fbEnvironmentZones 		: ARRAY[0..1] OF FB_SensorVirtual_Vaisala; 				// ARRAY[0..10] OF FB_SensorVirtual_Vaisala;
	fbLevelWaterControls 	: ARRAY[1..2] OF FB_LevelWaterControl; 
	
	nModbusUnitIDs: ARRAY[0..10] OF UINT := [11(0)];

	//fbHumidityControl 		: FB_BangBangControl;
	fbHumidityControl 		: FB_ControlLoop_PID;
	
	fbHumidityFilter:		FB_SigCond_MovingAverage := (nSamplesToFilter := 30, tCtrlCycleTime := T#2S, tTaskCycleTime := T#10MS);
	fbTON_HumMovAg: 		TON := (PT := T#2S, IN := FALSE);
	bResetTimer: 			BOOL := FALSE;
	
	fbCO2Control 			: FB_BangBangControl;
	//fbTemperatureControl 	: FB_BangBangControl_Analog;
	// fbTemperatureControl 	: FB_ControlLoop_HVAC;
	fbTemperatureControl 	: FB_ControlLoop_HVAC_1;
 
	fbFanControl_Exhaust:		FB_BangBangControl;	 
	fbFanControl_Circulation:	FB_BangBangControl;
	
	{attribute 'OPC.UA.DA' := '1'}
	rStackHumidity : REAL;
	{attribute 'OPC.UA.DA' := '1'}
	rStackCO2 : REAL;
	{attribute 'OPC.UA.DA' := '1'}
	rStackTemp : REAL;
	
	
END_VAR

IF bFirstRun THEN
	bFirstRun := FALSE;
	nModbusUnitIDs[0] := nSensorModbusID_1;
	nModbusUnitIDs[1] := nSensorModbusID_2;
	// nModbusUnitIDs[1] := nSensorModbusID_2; - bring this back after testing
	fbTON_HumMovAg(IN := TRUE);
	// run the temp and CO2 controls
	fbCO2Control.setState(E_DeviceState.RUNNING);
	fbTemperatureControl.setState(E_DeviceState.RUNNING);
	//fbHumidityControl.setState(E_DeviceState.RUNNING);

END_IF

IF bResetTimer THEN
	fbTON_HumMovAg(IN := TRUE);
	bResetTimer := FALSE;
END_IF

fbTON_HumMovAg();

(*
scanInputs();
*)

// Read temp, CO2 and humidity from Vaisala sensors
fbEnvironmentZones[0](nModbusUnitIDs := nModbusUnitIDs, rMaxDiscrepency := 0.1, fbModbusManager := fbModbusManager, sZoneName := sZoneName);
rStackCO2 		:= fbEnvironmentZones[0].rCO2; 
//rStackHumidity 	:= fbEnvironmentZones[0].rHumidity;
rStackTemp 		:= fbEnvironmentZones[0].rTemperature;

fbHumidityFilter();
// filter the humidity values
IF fbTON_HumMovAg.Q THEN
	fbHumidityFilter(fIn := fbEnvironmentZones[0].rHumidity);
	fbTON_HumMovAg(IN := FALSE);
	bResetTimer := TRUE;
	rStackHumidity	:= fbHumidityFilter.fOut;
END_IF

IF NOT stInputs.bParamsInitialised THEN
		fbLevelWaterControls[1].fbValve.enable();
		//fbLevelWaterControls[1].fbValve(bNO_or_NC_0_or_1 := stInputs.bIrrigatorValve_NC_1_NO_0);
		fbLevelWaterControls[1].fbValve();
		fbLevelWaterControls[1].fbValve.close();
		

END_IF

IF stInputs.bParamsInitialised THEN
	scanInputs();
	// control for humidity
	//fbHumidityControl(nProcessValue := rStackHumidity, sParameterName := 'Humidity', bEnabled := stInputs.HumidityControl.bEnabled);
	fbHumidityControl(nProcessValue := fbHumidityFilter.fOut, sParameterName := 'Humidity', bEnabled := stInputs.HumidityControl.bEnabled);
	// bang bang control for CO2
	fbCO2Control(rCurrentValue := rStackCO2, sParameterName := 'CO2', bEnabled := stInputs.CO2Control.bEnabled);
	// bang bang analog control for temperature
	fbTemperatureControl(rCurrentValue := rStackTemp, sParameterName := 'Temperature', nControlValue := ADR(stInputsHVAC.Setpoint), bEnabled := stInputs.TemperatureControl.bEnabled);
	//fbHumidityControl(rCurrentValue := rStackHumidity, sParameterName := 'Humidity', bEnabled := stInputs.HumidityControl.bEnabled);
	fbFanControl_Exhaust(rCurrentValue := rStackCO2, sParameterName := 'Exhaust Fan Control', bEnabled := stInputs.FanControl_Circulation.bEnabled);
	fbFanControl_Circulation(rCurrentValue := rStackCO2, sParameterName := 'Circulation Fan Control', bEnabled := stInputs.FanControl_Exhaust.bEnabled);
	FOR i := 1 TO nLevels DO
		// Irrigation valve
		fbLevelWaterControls[i](nLevel := i, stSCInputs := stInputs);
	END_FOR
END_IF

// Function blocks which have an instance for every level...


checkCropJobs();

METHOD checkCropJobs : BOOL
VAR_INPUT
END_VAR

// reset all crop jobs to false. Any active ones will be changed to true.

fbLevelWaterControls[1].bActiveCropJob := FALSE;


FOR i := 0 TO GVL.MaxCropJob DO
	
	// check if this crop job is coming FROM this stack
	IF Inputs.CropJobs[i].crop.stack = nStack AND Inputs.CropJobs[i].job_status > E_Job_Status.waiting AND Inputs.CropJobs[i].job_status < E_Job_Status.finished THEN
		fbLevelWaterControls[1].bActiveCropJob := TRUE;
	END_IF
	
	// check if this crop job is going TO this stack
	IF Inputs.CropJobs[i].stack = nStack AND Inputs.CropJobs[i].job_status > E_Job_Status.waiting AND Inputs.CropJobs[i].job_status < E_Job_Status.finished THEN
		fbLevelWaterControls[1].bActiveCropJob := TRUE;
	END_IF

END_FOR
END_METHOD

METHOD FB_init : BOOL
VAR_INPUT
	bInitRetains : BOOL; // if TRUE, the retain variables are initialized (warm start / cold start)
	bInCopyCode : BOOL;  // if TRUE, the instance afterwards gets moved into the copy code (online change)
	
	ID : STRING;
	Description : STRING;
	ModID_Sensor1: UINT;
	ModID_Sensor2: UINT;
	ZoneName:			STRING;
END_VAR

sID := ID;
sDescr := Description;

nSensorModbusID_1 := ModID_Sensor1;
nSensorModbusID_2 := ModID_Sensor2;
sZoneName := ZoneName;
END_METHOD

METHOD scanInputs : BOOL
VAR_INPUT
END_VAR



fbHumidityControl.bEnabled 				:= stInputs.HumidityControl.bEnabled;
fbHumidityControl.nAdjustDelay 			:= stInputs.HumidityControl.nAdjustDelay;
//fbHumidityControl.nAdjustDownDuration 	:= stInputs.HumidityControl.nAdjustDownDuration;
//fbHumidityControl.nAdjustUpDuration 	:= stInputs.HumidityControl.nAdjustUpDuration;
fbHumidityControl.rAlarmHigh 			:= stInputs.HumidityControl.rAlarmHigh;
fbHumidityControl.rAlarmLow 			:= stInputs.HumidityControl.rAlarmLow;
fbHumidityControl.rLimitHigh 			:= stInputs.HumidityControl.rLimitHigh;
fbHumidityControl.rLimitLow 			:= stInputs.HumidityControl.rLimitLow;

fbCO2Control.bEnabled 				:= stInputs.CO2Control.bEnabled;
fbCO2Control.nAdjustDelay 			:= stInputs.CO2Control.nAdjustDelay;
fbCO2Control.nAdjustDownDuration 	:= stInputs.CO2Control.nAdjustDownDuration;
fbCO2Control.nAdjustUpDuration 		:= stInputs.CO2Control.nAdjustUpDuration;
fbCO2Control.rAlarmHigh 			:= stInputs.CO2Control.rAlarmHigh;
fbCO2Control.rAlarmLow 				:= stInputs.CO2Control.rAlarmLow;
fbCO2Control.rLimitHigh 			:= stInputs.CO2Control.rLimitHigh;
fbCO2Control.rLimitLow 				:= stInputs.CO2Control.rLimitLow;

fbTEMPERATUREControl.bEnabled 				:= stInputs.TemperatureControl.bEnabled;
fbTEMPERATUREControl.nAdjustDelay 			:= stInputs.TemperatureControl.nAdjustDelay;
fbTEMPERATUREControl.nAdjustDownIncrement 	:= stInputs.TemperatureControl.nAdjustDownIncrement;
fbTEMPERATUREControl.nAdjustUpIncrement 	:= stInputs.TemperatureControl.nAdjustUpIncrement;
fbTEMPERATUREControl.rAlarmHigh 			:= stInputs.TemperatureControl.rAlarmHigh;
fbTEMPERATUREControl.rAlarmLow 				:= stInputs.TemperatureControl.rAlarmLow;
fbTEMPERATUREControl.rLimitHigh 			:= stInputs.TemperatureControl.rLimitHigh;
fbTEMPERATUREControl.rLimitLow 				:= stInputs.TemperatureControl.rLimitLow;

fbTemperatureControl.nDegPerHr				:= stInputs.TemperatureControl.rDegPerHr;
END_METHOD

END_FUNCTION_BLOCK

// ---- POUs/07 Systems/RND/FB_System_RND_HVAC.TcPOU
FUNCTION_BLOCK FB_System_RND_HVAC
VAR_IN_OUT
	// Hold a reference to MBMaster - may need to share this with other dosing machines if only 1 x RS485 card is used for both
	{attribute 'OPC.UA.DA' := '0'}
  	{attribute 'OPC.UA.DA.StructuredType' := '0'}
	fbModbusManager: 	FB_ModbusManager;    // We can read 32 registers using one query
END_VAR

VAR
	bFirstRun: BOOL := TRUE;
	bResetTimer: BOOL := TRUE;
	tgModReadAdaptorStatus: R_TRIG;
	
	
	nModbusID: INT := 1;
	nNumberHVACUnits: INT := 13;
	
	stModReadAdaptorStatus: 				ST_Modbus_ReadRequest;
	
	stModReadIndoorUnitConnStatus: 			ST_Modbus_ReadRequest;
	stModReadIndoorUnitCommsStatus: 		ST_Modbus_ReadRequest;
	stModReadIndoorUnitSetpoits: 			ARRAY[1..13] OF ST_Modbus_ReadRequest;
	stModReadIndoorUnitPower: 				ARRAY[1..13] OF ST_Modbus_ReadRequest;
	
	stModWriteaAdaptorStatus:				ST_Modbus_WriteRequest;
	stModWriteIndoorRoom:					ST_Modbus_WriteRequest;
	stModWriteIndoorSetpoint_R6:			ST_Modbus_WriteRequest;
	stModWriteIndoorSetpoint_R7:			ST_Modbus_WriteRequest;
	stModWriteIndoorSetpoint_R8:			ST_Modbus_WriteRequest;
	stModWriteIndoorSetpoint_R9:			ST_Modbus_WriteRequest;
	stModWriteIndoorControlPower:			ARRAY[1..13] OF ST_Modbus_WriteRequest;
	stModWriteIndoorControlSetpoint:		ARRAY[1..13] OF ST_Modbus_WriteRequest;
	
	bRoom7or9: BOOL := FALSE;
	nRoomNumber: UINT := 6;
	
	fbTON_DataRefresh: TON := (PT := T#1m, IN := FALSE);
	
	// delete this after commissioning (used for testing)
	modWrite: R_TRIG;
	stModWrite: ST_Modbus_WriteRequest;
	
		// delete this after commissioning (used for testing)
	modRead: 	R_TRIG;
	stModRead: 	ST_Modbus_ReadRequest;
END_VAR

VAR_OUTPUT
	{attribute 'OPC.UA.DA' := '1'}
  	{attribute 'OPC.UA.DA.StructuredType' := '1'}
	fbRND_HVAC: ARRAY[1..13] OF FB_HVAC_RND_Indoor_Unit;
	
	
	i: INT := 0;
	
END_VAR

IF bFirstRun THEN
	devices_init();
	bFirstRun := FALSE;
	initModRequests();
	
	fbModbusManager.addRequest_Write(WriteRequest := ADR(stModWriteaAdaptorStatus));
	fbModbusManager.addRequest_Write(WriteRequest := ADR(stModWriteIndoorRoom));
END_IF

IF bResetTimer THEN
	fbTON_DataRefresh(IN := TRUE);
	bResetTimer := FALSE;
END_IF

fbTON_DataRefresh();
scanInputs();

IF fbTON_DataRefresh.Q THEN
	//fbModbusManager.addRequest_Read(ReadRequest := ADR(stModReadAdaptorStatus));
	//fbModbusManager.addRequest_Read(ReadRequest := ADR(stModReadIndoorUnitConnStatus));
	//fbModbusManager.addRequest_Read(ReadRequest := ADR(stModReadIndoorUnitCommsStatus));
	CASE nRoomNumber OF
		6:
			stModWriteIndoorSetpoint_R6.WriteRegVals[1] := INT_TO_WORD(REAL_TO_INT(Inputs.HVAC_RND[6].Setpoint * 10));
			fbModbusManager.addRequest_Write(WriteRequest := ADR(stModWriteIndoorSetpoint_R6));		
			nRoomNumber := 7;
	
		7:
			stModWriteIndoorSetpoint_R7.WriteRegVals[1] := INT_TO_WORD(REAL_TO_INT(Inputs.HVAC_RND[7].Setpoint * 10));
			fbModbusManager.addRequest_Write(WriteRequest := ADR(stModWriteIndoorSetpoint_R7));
			nRoomNumber := 8;
			
		8:
			stModWriteIndoorSetpoint_R8.WriteRegVals[1] := INT_TO_WORD(REAL_TO_INT(Inputs.HVAC_RND[8].Setpoint * 10));
			fbModbusManager.addRequest_Write(WriteRequest := ADR(stModWriteIndoorSetpoint_R8));
			nRoomNumber := 9;	
		
		9:
			stModWriteIndoorSetpoint_R9.WriteRegVals[1] := INT_TO_WORD(REAL_TO_INT(Inputs.HVAC_RND[9].Setpoint * 10));
			fbModbusManager.addRequest_Write(WriteRequest := ADR(stModWriteIndoorSetpoint_R9));
			nRoomNumber := 6;		
			
	END_CASE
	
	(*
	IF bRoom7or9 THEN
			stModWriteIndoorSetpoint_R7.WriteRegVals[1] := INT_TO_WORD(REAL_TO_INT(Inputs.HVAC_RND[7].Setpoint * 10));
			fbModbusManager.addRequest_Write(WriteRequest := ADR(stModWriteIndoorSetpoint_R7));
			bRoom7or9 := FALSE;
	ELSE
			stModWriteIndoorSetpoint_R9.WriteRegVals[1] := INT_TO_WORD(REAL_TO_INT(Inputs.HVAC_RND[9].Setpoint * 10));
			fbModbusManager.addRequest_Write(WriteRequest := ADR(stModWriteIndoorSetpoint_R9));
			bRoom7or9 := TRUE;
	END_IF
	*)

	

	
	//FOR i := 1 TO 13 DO
		//fbModbusManager.addRequest_Read(ReadRequest := ADR(stModReadIndoorUnitSetpoits[i]));
		//fbModbusManager.addRequest_Read(ReadRequest := ADR(stModReadIndoorUnitPower[i]));
		//fbModbusManager.addRequest_Write(WriteRequest := ADR(stModWriteIndoorControlPower));
		//fbModbusManager.addRequest_Write(WriteRequest := ADR(stModWriteIndoorControlSetpoint));
	//END_FOR
	
	fbTON_DataRefresh(IN := FALSE);
	bResetTimer := TRUE;
END_IF


modRead();
IF modRead.Q THEN
	fbModbusManager.addRequest_Read_Priority(ReadRequest := ADR(stModRead));
END_IF


modWrite();
IF modWrite.Q THEN
	fbModbusManager.addRequest_Write(WriteRequest := ADR(stModWrite));
END_IF

devices_update();

METHOD devices_init : BOOL
VAR_INPUT
END_VAR
(*
aHVAC_IndoorUnits[1] := ADR(fbRND1_HVAC);
aHVAC_IndoorUnits[2] := ADR(fbRND2_HVAC);
aHVAC_IndoorUnits[3] := ADR(fbRND3_HVAC);
aHVAC_IndoorUnits[4] := ADR(fbRND4_HVAC);
aHVAC_IndoorUnits[5] := ADR(fbRND5_HVAC);
aHVAC_IndoorUnits[6] := ADR(fbRND6_HVAC);
aHVAC_IndoorUnits[7] := ADR(fbRND7_HVAC);
aHVAC_IndoorUnits[8] := ADR(fbRND8_HVAC);
aHVAC_IndoorUnits[9] := ADR(fbRND9_HVAC);
aHVAC_IndoorUnits[10] := ADR(fbRND10_HVAC);
aHVAC_IndoorUnits[11] := ADR(fbRND11_HVAC);
aHVAC_IndoorUnits[12] := ADR(fbRND12_HVAC);

*)
END_METHOD

METHOD devices_update : BOOL
VAR_INPUT
END_VAR
(*
FOR i := 1 TO 13 DO
	fbRND_HVAC[i].bOnOff_1_0 := 	stModReadIndoorUnitPower[i].ReadRegsVals[1].0;
	fbRND_HVAC[1].nSetpoint_RO := 	WORD_TO_REAL(stModReadIndoorUnitSetpoits[i].ReadRegsVals[1])/10;
	
END_FOR

fbRND_HVAC[1].bConnectionStatus := stModReadIndoorUnitConnStatus.ReadRegsVals[1].0;
fbRND_HVAC[2].bConnectionStatus := stModReadIndoorUnitConnStatus.ReadRegsVals[1].1;
fbRND_HVAC[3].bConnectionStatus := stModReadIndoorUnitConnStatus.ReadRegsVals[1].2;
fbRND_HVAC[4].bConnectionStatus := stModReadIndoorUnitConnStatus.ReadRegsVals[1].3;
fbRND_HVAC[5].bConnectionStatus := stModReadIndoorUnitConnStatus.ReadRegsVals[1].4;
fbRND_HVAC[6].bConnectionStatus := stModReadIndoorUnitConnStatus.ReadRegsVals[1].5;
fbRND_HVAC[7].bConnectionStatus := stModReadIndoorUnitConnStatus.ReadRegsVals[1].6;
fbRND_HVAC[8].bConnectionStatus := stModReadIndoorUnitConnStatus.ReadRegsVals[1].7;
fbRND_HVAC[9].bConnectionStatus := stModReadIndoorUnitConnStatus.ReadRegsVals[1].8;
fbRND_HVAC[10].bConnectionStatus := stModReadIndoorUnitConnStatus.ReadRegsVals[1].9;
fbRND_HVAC[11].bConnectionStatus := stModReadIndoorUnitConnStatus.ReadRegsVals[1].10;
fbRND_HVAC[12].bConnectionStatus := stModReadIndoorUnitConnStatus.ReadRegsVals[1].11;
fbRND_HVAC[13].bConnectionStatus := stModReadIndoorUnitConnStatus.ReadRegsVals[1].12;

fbRND_HVAC[1].bCommsStatus := stModReadIndoorUnitCommsStatus.ReadRegsVals[1].0;
fbRND_HVAC[2].bCommsStatus := stModReadIndoorUnitCommsStatus.ReadRegsVals[1].1;
fbRND_HVAC[3].bCommsStatus := stModReadIndoorUnitCommsStatus.ReadRegsVals[1].2;
fbRND_HVAC[4].bCommsStatus := stModReadIndoorUnitCommsStatus.ReadRegsVals[1].3;
fbRND_HVAC[5].bCommsStatus := stModReadIndoorUnitCommsStatus.ReadRegsVals[1].4;
fbRND_HVAC[6].bCommsStatus := stModReadIndoorUnitCommsStatus.ReadRegsVals[1].5;
fbRND_HVAC[7].bCommsStatus := stModReadIndoorUnitCommsStatus.ReadRegsVals[1].6;
fbRND_HVAC[8].bCommsStatus := stModReadIndoorUnitCommsStatus.ReadRegsVals[1].7;
fbRND_HVAC[9].bCommsStatus := stModReadIndoorUnitCommsStatus.ReadRegsVals[1].8;
fbRND_HVAC[10].bCommsStatus := stModReadIndoorUnitCommsStatus.ReadRegsVals[1].9;
fbRND_HVAC[11].bCommsStatus := stModReadIndoorUnitCommsStatus.ReadRegsVals[1].10;
fbRND_HVAC[12].bCommsStatus := stModReadIndoorUnitCommsStatus.ReadRegsVals[1].11;
fbRND_HVAC[13].bCommsStatus := stModReadIndoorUnitCommsStatus.ReadRegsVals[1].12;
*)
END_METHOD

METHOD FB_init : BOOL
VAR_INPUT
	bInitRetains : BOOL; // if TRUE, the retain variables are initialized (warm start / cold start)
	bInCopyCode : BOOL;  // if TRUE, the instance afterwards gets moved into the copy code (online change)
	
	ModbusID: UINT;
END_VAR
nModbusID := ModbusID;
END_METHOD

METHOD initModRequests : BOOL
VAR_INPUT
END_VAR

stModReadAdaptorStatus.SlaveAddress := 1;
stModReadAdaptorStatus.AdrFirstSlaveRegisterRead := 0;
stModReadAdaptorStatus.QtyWordsToRead := 1;

stModReadIndoorUnitConnStatus.SlaveAddress := 1;
stModReadIndoorUnitConnStatus.AdrFirstSlaveRegisterRead := 1;
stModReadIndoorUnitConnStatus.QtyWordsToRead := 1;

stModReadIndoorUnitCommsStatus.SlaveAddress := 1;
stModReadIndoorUnitCommsStatus.AdrFirstSlaveRegisterRead := 5;
stModReadIndoorUnitCommsStatus.QtyWordsToRead := 1;

stModWriteaAdaptorStatus.SlaveAddress := 1;
stModWriteaAdaptorStatus.AdrFirstSlaveRegisterWrite := 1;
stModWriteaAdaptorStatus.QtyWordsToWrite := 1;
stModWriteaAdaptorStatus.WriteRegVals[1] := 32768; // turn modbus comms on

stModWriteIndoorRoom.SlaveAddress := 1;
stModWriteIndoorRoom.AdrFirstSlaveRegisterWrite := 2018;
stModWriteIndoorRoom.QtyWordsToWrite := 1;
stModWriteIndoorRoom.WriteRegVals[1] := 1889;

stModWriteIndoorSetpoint_R6.SlaveAddress := 1;
stModWriteIndoorSetpoint_R6.AdrFirstSlaveRegisterWrite := 2017;
stModWriteIndoorSetpoint_R6.QtyWordsToWrite := 1;

stModWriteIndoorSetpoint_R7.SlaveAddress := 1;
stModWriteIndoorSetpoint_R7.AdrFirstSlaveRegisterWrite := 2020;
stModWriteIndoorSetpoint_R7.QtyWordsToWrite := 1;

stModWriteIndoorSetpoint_R8.SlaveAddress := 1;
stModWriteIndoorSetpoint_R8.AdrFirstSlaveRegisterWrite := 2023;
stModWriteIndoorSetpoint_R8.QtyWordsToWrite := 1;

stModWriteIndoorSetpoint_R9.SlaveAddress := 1;
stModWriteIndoorSetpoint_R9.AdrFirstSlaveRegisterWrite := 2026;
stModWriteIndoorSetpoint_R9.QtyWordsToWrite := 1;


FOR i := 1 TO nNumberHVACUnits DO
	stModReadIndoorUnitSetpoits[i].SlaveAddress := 1;
	stModReadIndoorUnitSetpoits[i].AdrFirstSlaveRegisterRead := 2002 + ((i-1) * 6);
	stModReadIndoorUnitSetpoits[i].QtyWordsToRead := 1;
	
	stModReadIndoorUnitPower[i].SlaveAddress := 1;
	stModReadIndoorUnitPower[i].AdrFirstSlaveRegisterRead := 2000 + ((i-1) * 6);
	stModReadIndoorUnitPower[i].QtyWordsToRead := 1;
	
	stModWriteIndoorControlPower[i].SlaveAddress := 1;
	stModWriteIndoorControlPower[i].AdrFirstSlaveRegisterWrite := 2000 + ((i-1)*3);
	stModWriteIndoorControlPower[i].QtyWordsToWrite := 1;
	
	stModWriteIndoorControlSetpoint[i].SlaveAddress := 1;
	stModWriteIndoorControlSetpoint[i].AdrFirstSlaveRegisterWrite := 2002 + + ((i-1)*3);
	stModWriteIndoorControlSetpoint[i].QtyWordsToWrite := 1;
	
END_FOR
END_METHOD

METHOD scanInputs : BOOL
VAR_INPUT
END_VAR
FOR i := 1 TO nNumberHVACUnits DO
	IF Inputs.HVAC_RND[i].Power THEN
		stModWriteIndoorControlPower[i].WriteRegVals[1] := 1;
	ELSE
		stModWriteIndoorControlPower[i].WriteRegVals[1] := 0;
	END_IF
	//stModWriteIndoorControlPower[i].WriteRegVals[1] := BOOL_TO_WORD(Inputs.HVAC_RND[i].Power);
	stModWriteIndoorControlSetpoint[i].WriteRegVals[1] := (REAL_TO_INT(Inputs.HVAC_RND[i].Setpoint * 10.0));
	// stModWriteIndoorControlPower[i].WriteRegVals[i] := 2#0111001001100000 AND stModWriteIndoorControlPower[i].WriteRegVals[i]; // binary word includes mandatory fields (fan power / volume / control)
END_FOR
END_METHOD

END_FUNCTION_BLOCK

// ---- POUs/06 Machines/_ss/FB_Machine_DosingMachine_TEST2.TcPOU
{attribute 'OPC.UA.DA.StructuredType' := '1'}
FUNCTION_BLOCK FB_Machine_DosingMachine_TEST2 EXTENDS FB_BaseMachine

VAR
	
	// Set limits for machines 
	// Bag filter differential pressures
	nPressureDiffLimit_Filter1_Limit: REAL := 6000; //kpa
	nPressureDiffLimit_Filter2_Limit: REAL := 6000; //kpa
	
	// Dosing / Nutrient Limits & SetPoints
	nEC_Low_Limit: REAL := 1000;
	nEC_High_Limit: REAL := 1400;
	nEC_SetPoint: REAL := 1200;
	
	nPH_Low_Limit: REAL := 7.8;
	nPH_High_Limit: REAL := 8.0;
	nPH_SetPoint: REAL := 8.2;
	
	nDO_Low_Limit: REAL := 500;
	nDO_High_Limit: REAL := 700;
	nDO_SetPoint: REAL := 600;
	
	nORP_Low_Limit: REAL := 1000;
	nORP_High_Limit: REAL := 1200;
	nORP_SetPoint: REAL := 1400;
	
	nTemp_Low_Limit: REAL  := 1.5;
	nTemp_High_Limit: REAL := 26;
	nTemp_SetPoint: REAL := 18;  // not applicable for now
	
	
	//Sequence Manager & Sequences
	fbSequenceManager: FB_SequenceManager;
	
	{attribute 'OPC.UA.DA' := '0'} 
	fbSeqDMMain: FB_SequenceDM_Main;
	{attribute 'OPC.UA.DA' := '0'} 
	fbSeqDMCal: FB_SequenceDM_Calibrate;
	{attribute 'OPC.UA.DA' := '0'} 
	fbSeqDMFill: FB_SequenceDM_Fill;
	{attribute 'OPC.UA.DA' := '0'} 
	fbSeqDMDrain: FB_SequenceDM_Drain;
	
	
	// Hold a reference to MBMaster - may need to share this with other dosing machines if only 1 x RS485 card is used for both
	{attribute 'OPC.UA.DA' := '0'} 
	fbModbusMaster: REFERENCE TO FB_ModbusMaster;
	
	// Hold a reference to these tanks (they are shared between dosing machines and water treatment)
	fbTank_pHUP: REFERENCE TO FB_Tank;
	fbTank_pHDown: REFERENCE TO FB_Tank;
	fbTank_NutrientA: REFERENCE TO FB_Tank;
	fbTank_NutrientB: REFERENCE TO FB_Tank;
	fbTank_NutrientC: REFERENCE TO FB_Tank;

	// Dosing Pumps
	fbDosingPump_phUp		: FB_DosingPumpPRISMA(MotorID:= '_DP1', MotorDescr:= ' Dosing Pump - pH Up' , ModbusUnitID:=2 , ModbusMaster:=fbModbusMaster);
	fbDosingPump_phDown		: FB_DosingPumpPRISMA(MotorID:= '_DP2', MotorDescr:= ' Dosing Pump - pH Down' , ModbusUnitID:=3 , ModbusMaster:=fbModbusMaster);
	fbDosingPump_NutrientA	: FB_DosingPumpPRISMA(MotorID:= '_DP3', MotorDescr:= ' Dosing Pump - Nutrient A' , ModbusUnitID:=4 , ModbusMaster:=fbModbusMaster);	
	fbDosingPump_NutrientB	: FB_DosingPumpPRISMA(MotorID:= '_DP4', MotorDescr:= ' Dosing Pump - Nutrient B' , ModbusUnitID:=5 , ModbusMaster:=fbModbusMaster);
	fbDosingPump_NutrientC	: FB_DosingPumpPRISMA(MotorID:= '_DP5', MotorDescr:= ' Dosing Pump - Nutrient C' , ModbusUnitID:=6 , ModbusMaster:=fbModbusMaster);
	
	
	// Atlas Sensors
	fbSensor_DissOx1: FB_Sensor_AtlasDO(SensorID:= '-SU1-DO1' , SensorDescr:= ' Dissolved Oxygen - Sensor 1', SensorType:= E_SensorType.Analogue);
	fbSensor_DissOx2: FB_Sensor_AtlasDO(SensorID:= '-SU1-DO2' , SensorDescr:= ' Dissolved Oxygen - Sensor 2', SensorType:= E_SensorType.Analogue);
	fbSensor_DissOx: FB_DualRedundantSensor(SensorID:= 'SU1-DO', SensorDescr:= 'Dissolved Oxygen Sensing', SensorType:= E_SensorType.Analogue);
	//fbSensor_DissOx.addSensors(Sensor1 := fbSensor_DissOx1, Sensor2 := fbSensor_DissOx2);
	
	
	fbSensor_EC1: FB_Sensor_AtlasEC(SensorID:= '-SU1-EC1', SensorDescr:= ' Electrical Conductivity - Sensor 1', SensorType:= E_SensorType.Analogue);
	fbSensor_EC2: FB_Sensor_AtlasEC(SensorID:= '-SU1-EC2', SensorDescr:= ' Electrical Conductivity - Sensor 2', SensorType:= E_SensorType.Analogue);
	fbSensor_EC: FB_DualRedundantSensor(SensorID:= 'SU1-EC', SensorDescr:= 'Electrical Conductivity Sensing',  SensorType:= E_SensorType.Analogue);
	
	fbSensor_ORP1: FB_Sensor_AtlasORP(SensorID:= '-SU1-ORP1', SensorDescr:= ' Oxidation / Reduction Potential - Sensor 1', SensorType:= E_SensorType.Analogue);
	fbSensor_ORP2: FB_Sensor_AtlasORP(SensorID:= '-SU1-ORP2', SensorDescr:= ' Oxidation / Reduction Potential - Sensor 2', SensorType:= E_SensorType.Analogue);
	fbSensor_ORP: FB_DualRedundantSensor(SensorID:= 'SU1-ORP', SensorDescr:= 'Oxidation / Reduction Potential', SensorType:= E_SensorType.Analogue);
	
	fbSensor_PH1: FB_Sensor_AtlasPH(SensorID:= '-SU1-PH1', SensorDescr:= ' Potential Hydrogen (ph) - Sensor 1', SensorType:= E_SensorType.Analogue);
	fbSensor_PH2: FB_Sensor_AtlasPH(SensorID:= '-SU1-PH2', SensorDescr:= ' Potential Hydrogen (ph) - Sensor 2', SensorType:= E_SensorType.Analogue);
	fbSensor_PH: FB_DualRedundantSensor(SensorID:= 'SU1-PH', SensorDescr:= 'Potential Hydrogen (ph)', SensorType:= E_SensorType.Analogue);
		
	fbSensor_TMP1: FB_Sensor_AtlasTEMP(SensorID:= '-SU1-TMP1', SensorDescr:= 'Water Temperature - Sensor 1', SensorType:= E_SensorType.Analogue);
	fbSensor_TMP2: FB_Sensor_AtlasTEMP(SensorID:= '-SU1-TMP2', SensorDescr:= 'Water Temperature - Sensor 2', SensorType:= E_SensorType.Analogue);
	fbSensor_TMP: FB_DualRedundantSensor(SensorID:= 'SU1-TMP', SensorDescr:= 'Water Temperature', SensorType:= E_SensorType.Analogue);
	
	fbSensor_SumpLIT1 : FB_Sensor_4_20mA_Generic(SensorID:= '_SU1_LIT1', SensorDescr:= ' Sump Level Transmitter 1' , SensorType:= E_SensorType.Analogue); 
	fbSensor_FilterPIT1: FB_Sensor_OceanControlsPressureTx_BVS006NA( SensorID:= '_SU1_PIT1',	SensorDescr:= ' Bag Filter Pressure Sensor 1', SensorType:= E_SensorType.Analogue);
	fbSensor_FilterPIT2: FB_Sensor_OceanControlsPressureTx_BVS006NA( SensorID:= '_SU1_PIT2',	SensorDescr:= ' Bag Filter Pressure Sensor 2', SensorType:= E_SensorType.Analogue);
	fbSensor_FilterPIT3: FB_Sensor_OceanControlsPressureTx_BVS006NA( SensorID:= '_SU1_PIT3',	SensorDescr:= ' Bag Filter Pressure Sensor 3', SensorType:= E_SensorType.Analogue);  
	fbSensor_DosingPIT1: FB_Sensor_OceanControlsPressureTx_BVS006NA( SensorID:= '_SU1_PIT4',	SensorDescr:= 'Dosing Line Pressure Transmitter', SensorType:= E_SensorType.Analogue);
	
	// Actuated Valves
	fbValve_DosingSupply: FB_Valve_ONOFF_woMonitoring(ValveID:= '_SU1_V1', ValveDescr:= ' Dosing Circuit Supply Valve' ); 
	fbValve_IrrigatorSupply: FB_Valve_ONOFF_woMonitoring(ValveID:= '_SU1_V2', ValveDescr:= ' Irrigator Supply Valve' ); 
	fbValve_WasteWaterReturn: FB_Valve_ONOFF_woMonitoring(ValveID:= '_SU1_V4', ValveDescr:= ' Waste Water Return Valve');
	
	// Vendor Units	
	fbUnit_OxyInjector: FB_OxygenInjector(UnitID:= '_SU1_OXY1' , UnitDescr:= ' Oxygen Injector');	 
	fbUnit_UltraSonCleaner: FB_UltraSonicCleaner(UnitID:= '_SU1_USC1' , UnitDescr:= ' Ultrasonic Cleaner');
	
	// VSD Pumps
	fbPump_MainPumpA: FB_PumpVSD_DanfossFC202(PumpID:='_SU1_PU1_A' , PumpDescr:=' Main Pump - A');	 
	fbPump_MainPumpB: FB_PumpVSD_DanfossFC202(PumpID:='_SU1_PU1_B' , PumpDescr:=' Main Pump - B');	 
	fbDrumFilter1: FB_DrumFilter_Faivre120(FilterID:= '_SU1_DF1' , FIlterDescr:= ' Drum Filter');	 
	fbUVFilter1: FB_UVFilter_UltraAqua_MR4_220PP(UnitID:= '_SU1_UVC1', UnitDescr:= ' Ultraviolet Filter' );	 
	
	// Passive Components
	fbBagFilter1: FB_BagFilter(FilterID:= 'SU1-FTR1', FilterDescr:= 'Dosing Sump Bag Filter 1' , DiffPress_Upstream:= fbSensor_FilterPIT1, DiffPress_Downstream:= fbSensor_FilterPIT2);
	fbBagFilter2: FB_BagFilter(FilterID:= 'SU1-FTR2', FilterDescr:= 'Dosing Sump Bag Filter 2' , DiffPress_Upstream:= fbSensor_FilterPIT2, DiffPress_Downstream:= fbSensor_FilterPIT3);
	fbSumpDosing: FB_Tank(TankID:= 'SU1', TankDescr:= 'Dosing Sump'); //, Sensor_LL:= fbSensor_SumpLIT1,Sensor_L:= fbSensor_SumpLIT1, Sensor_H:= fbSensor_SumpLIT1, Sensor_HH:= fbSensor_SumpLIT1,	Sensor_LIT:= fbSensor_SumpLIT1); 
	
	
	// Control Loops
	(*fbControlLoop_Dosing: FB_ControlLoop_Dosing(
								DosingPump_phUp := fbDosingPump_phUp, 
								DosingPump_phDOwn := fbDosingPump_phDown, 
								DosingPump_Nutrient_A := fbDosingPump_NutrientA, 
								DosingPump_Nutrient_B := fbDosingPump_NutrientB, 
								DosingPump_Nutrient_C := fbDosingPump_NutrientC, 
								Sensor_EC := fbSensor_EC, 
								Sensor_DO := fbSensor_DissOx, 
								Sensor_ORP := fbSensor_ORP, 
								Sensor_PH := fbSensor_PH, 
								Sensor_TEMP := fbSensor_TMP);
								*)
	
	
	
	// Package all components into structure to pass to sub-FBs 
	// This ST is populated by calling the populateComponents method
	{attribute 'OPC.UA.DA' := '0'} 
	stAllComponents: ST_DMComponents;
	
	
	
END_VAR

// Assign Pressure Sensors to Bag Filters & Tanks
fbBagFilter1.setPressureLimits();
fbBagFilter2.setPressureLimits();
//fbSumpDosing.setLevelSensors();

// Run Sequences
checkRunPermissives();

fbSequenceManager();

// Look for inputs


//Run Control Loops

// Cycle Through Device FBs
fbDosingPump_phUp();
fbDosingPump_phDown();
fbDosingPump_NutrientA();
fbDosingPump_NutrientB();
fbDosingPump_NutrientC();
fbSensor_DissOx1();
fbSensor_DissOx2();
fbSensor_EC1();
fbSensor_EC2();
fbSensor_ORP1();
fbSensor_ORP2();
fbSensor_PH1();
fbSensor_PH2();
fbSensor_TMP1();
fbSensor_TMP2();
fbSensor_SumpLIT1();
fbSensor_FilterPIT1();
fbSensor_FilterPIT2();
fbSensor_FilterPIT3();
fbValve_DosingSupply();
fbValve_IrrigatorSupply();
fbValve_WasteWaterReturn();
fbUnit_OxyInjector();
fbUnit_UltraSonCleaner();
fbPump_MainPumpA(); 
fbPump_MainPumpB();	 
fbDrumFilter1();	 
fbUVFilter1();	 
fbBagFilter1();
fbBagFilter2();
fbSumpDosing();

METHOD checkRunPermissive_DosingPump_NutrientA : BOOL
VAR_INPUT
END_VAR

VAR
	
END_VAR

IF fbSensor_DosingPIT1.getState() = E_DeviceState.OUT_OF_RANGE OR
	fbDosingPump_NutrientB.getState() = E_DeviceState.RUNNING OR
	fbDosingPump_NutrientC.getState() = E_DeviceState.RUNNING OR
	fbDosingPump_phUp.getState() = E_DeviceState.RUNNING OR
	fbDosingPump_phDown.getState() = E_DeviceState.RUNNING  THEN
	
		checkRunPermissive_DosingPump_NutrientA := FALSE;

ELSE
		checkRunPermissive_DosingPump_NutrientA := TRUE;
END_IF
END_METHOD

METHOD checkRunPermissive_DosingPump_NutrientB : BOOL
VAR_INPUT
END_VAR

IF fbSensor_DosingPIT1.getState() = E_DeviceState.OUT_OF_RANGE OR
	fbDosingPump_NutrientA.getState() = E_DeviceState.RUNNING OR
	fbDosingPump_NutrientC.getState() = E_DeviceState.RUNNING OR
	fbDosingPump_phUp.getState() = E_DeviceState.RUNNING OR
	fbDosingPump_phDown.getState() = E_DeviceState.RUNNING  THEN
	
		checkRunPermissive_DosingPump_NutrientB := FALSE;

ELSE
		checkRunPermissive_DosingPump_NutrientB := TRUE;
END_IF
END_METHOD

METHOD checkRunPermissive_DosingPump_NutrientC : BOOL
VAR_INPUT
END_VAR

IF fbSensor_DosingPIT1.getState() = E_DeviceState.OUT_OF_RANGE OR
	fbDosingPump_NutrientA.getState() = E_DeviceState.RUNNING OR
	fbDosingPump_NutrientB.getState() = E_DeviceState.RUNNING OR
	fbDosingPump_phUp.getState() = E_DeviceState.RUNNING OR
	fbDosingPump_phDown.getState() = E_DeviceState.RUNNING  THEN
	
		checkRunPermissive_DosingPump_NutrientC := FALSE;

ELSE
		checkRunPermissive_DosingPump_NutrientC := TRUE;
END_IF
END_METHOD

METHOD checkRunPermissive_DosingPump_phDown : BOOL
VAR_INPUT
END_VAR

IF fbSensor_DosingPIT1.getState() = E_DeviceState.OUT_OF_RANGE OR
	fbDosingPump_NutrientA.getState() = E_DeviceState.RUNNING OR
	fbDosingPump_NutrientB.getState() = E_DeviceState.RUNNING OR
	fbDosingPump_NutrientC.getState() = E_DeviceState.RUNNING OR
	fbDosingPump_phUp.getState() = E_DeviceState.RUNNING  THEN
	
		checkRunPermissive_DosingPump_phDown := FALSE;

ELSE
		checkRunPermissive_DosingPump_phDown := TRUE;
END_IF
END_METHOD

METHOD checkRunPermissive_DosingPump_phUp : BOOL
VAR_INPUT
END_VAR

IF fbSensor_DosingPIT1.getState() = E_DeviceState.OUT_OF_RANGE OR
	fbDosingPump_NutrientA.getState() = E_DeviceState.RUNNING OR
	fbDosingPump_NutrientB.getState() = E_DeviceState.RUNNING OR
	fbDosingPump_NutrientC.getState() = E_DeviceState.RUNNING OR
	fbDosingPump_phDown.getState() = E_DeviceState.RUNNING  THEN
	
		checkRunPermissive_DosingPump_phUp := FALSE;

ELSE
		checkRunPermissive_DosingPump_phUp := TRUE;
END_IF
END_METHOD

METHOD checkRunPermissive_OxyInjector : BOOL
VAR_INPUT
END_VAR

IF fbSumpDosing.getState() = E_DeviceState.OUT_OF_RANGE THEN

		checkRunPermissive_OxyInjector := FALSE;
ELSE
		checkRunPermissive_OxyInjector := TRUE;
END_IF
END_METHOD

METHOD checkRunPermissive_PumpMainPumpA : BOOL
VAR_INPUT
END_VAR

IF fbPump_MainPumpB.getState() = E_DeviceState.RUNNING OR
	(fbValve_IrrigatorSupply.getState() = E_DeviceState.CLOSED AND
		fbValve_WasteWaterReturn.getState() = E_DeviceState.CLOSED AND
		fbSensor_DosingPIT1.getState() = E_DeviceState.LOW_LOW) OR
	fbSumpDosing.getState() = E_DeviceState.LOW_LOW OR
	fbBagFilter1.getDiffPressure() > nPressureDiffLimit_Filter1_Limit OR
	fbBagFilter2.getDiffPressure() > nPressureDiffLimit_Filter2_Limit THEN
	
		checkRunPermissive_PumpMainPumpA := FALSE;
ELSE
	checkRunPermissive_PumpMainPumpA := TRUE;
END_IF
END_METHOD

METHOD checkRunPermissive_PumpMainPumpB : BOOL
VAR_INPUT
END_VAR

IF fbPump_MainPumpA.getState() = E_DeviceState.RUNNING OR
	(fbValve_IrrigatorSupply.getState() = E_DeviceState.CLOSED AND
		fbValve_WasteWaterReturn.getState() = E_DeviceState.CLOSED AND
		fbSensor_DosingPIT1.getState() = E_DeviceState.LOW_LOW) OR
	fbSumpDosing.getState() = E_DeviceState.LOW_LOW OR
	fbBagFilter1.getDiffPressure() > nPressureDiffLimit_Filter1_Limit OR
	fbBagFilter2.getDiffPressure() > nPressureDiffLimit_Filter2_Limit THEN
	
		checkRunPermissive_PumpMainPumpB := FALSE;
ELSE
	checkRunPermissive_PumpMainPumpB := TRUE;
END_IF
END_METHOD

METHOD checkRunPermissive_UltraSonCleaner : BOOL
VAR_INPUT
END_VAR

IF fbSumpDosing.getState() = E_DeviceState.LOW_LOW THEN
	
	checkRunPermissive_UltraSonCleaner := FALSE;
ELSE
	checkRunPermissive_UltraSonCleaner := TRUE;
END_IF
END_METHOD

METHOD checkRunPermissive_UVFilter : BOOL
VAR_INPUT
END_VAR


IF fbSumpDosing.getState() = E_DeviceState.LOW_LOW THEN
	checkRunPermissive_UVFilter := TRUE;
ELSE
	checkRunPermissive_UVFilter := FALSE;
END_IF
END_METHOD

METHOD checkRunPermissive_ValveIrrigatorSupply : BOOL
VAR_INPUT
END_VAR

// No interlocks exist for this valve 
IF FALSE THEN
	checkRunPermissive_ValveIrrigatorSupply := FALSE;
ELSE
	checkRunPermissive_ValveIrrigatorSupply := TRUE;
END_IF
END_METHOD

METHOD checkRunPermissive_ValveWasteWaterReturn : BOOL
VAR_INPUT
END_VAR

IF FALSE THEN
	checkRunPermissive_ValveWasteWaterReturn := FALSE;
ELSE
	checkRunPermissive_ValveWasteWaterReturn := TRUE;
END_IF
END_METHOD

METHOD checkRunPermissives : BOOL
VAR_INPUT
END_VAR
// Check RUN interlocks and stop motors / pumps & close / open valves

IF checkRunPermissive_DosingPump_phUp() <> TRUE THEN
	fbDosingPump_phUp.setOFF(RequestComplete := NULL);
END_IF

IF checkRunPermissive_DosingPump_phDown() <> TRUE THEN
	fbDosingPump_phDown.setOFF(RequestComplete := NULL);
END_IF

IF checkRunPermissive_DosingPump_NutrientA() <> TRUE THEN
	fbDosingPump_NutrientA.setOFF(RequestComplete := NULL);
END_IF

IF checkRunPermissive_DosingPump_NutrientB() <> TRUE THEN
	fbDosingPump_NutrientB.setOFF(RequestComplete := NULL);
END_IF

IF checkRunPermissive_DosingPump_NutrientC() <> TRUE THEN
	fbDosingPump_NutrientC.setOFF(RequestComplete := NULL);
END_IF

IF checkRunPermissive_OxyInjector() <> TRUE THEN
	fbUnit_OxyInjector.setOff();
END_IF

IF checkRunPermissive_PumpMainPumpA() <> TRUE THEN
	fbPump_MainPumpA.setReference(RefSetPoint := 0);
	// fbPump_MainPumpA.setOff(); check if this is needed when testing pump
END_IF

IF checkRunPermissive_PumpMainPumpB() <> TRUE THEN
	fbPump_MainPumpB.setReference(RefSetPoint := 0);
	// fbPump_MainPumpB.setOff(); check if this is needed when testing pump
END_IF

IF checkRunPermissive_UltraSonCleaner() <> TRUE THEN
	fbUnit_UltraSonCleaner.setOff();
END_IF

IF checkRunPermissive_UVFilter() <> TRUE THEN
	fbUVFilter1.setOff();
END_IF

IF checkRunPermissive_ValveIrrigatorSupply() <> TRUE THEN
	fbValve_IrrigatorSupply.close();
END_IF

IF checkStartPermissive_ValveWasteWaterReturn() <> TRUE THEN
	fbValve_WasteWaterReturn.close();
END_IF
END_METHOD

METHOD checkStartPermissive_DosingPump_NutrientA : BOOL
VAR_INPUT
END_VAR

IF fbSensor_DosingPIT1.getState() = E_DeviceState.OUT_OF_RANGE OR
	fbDosingPump_NutrientB.getState() = E_DeviceState.RUNNING OR
	fbDosingPump_NutrientC.getState() = E_DeviceState.RUNNING OR
	fbDosingPump_phUp.getState() = E_DeviceState.RUNNING OR
	fbDosingPump_phDown.getState() = E_DeviceState.RUNNING  THEN
	
		checkStartPermissive_DosingPump_NutrientA := FALSE;

ELSE
		checkStartPermissive_DosingPump_NutrientA := TRUE;
END_IF
END_METHOD

METHOD checkStartPermissive_DosingPump_NutrientB : BOOL
VAR_INPUT
END_VAR

IF fbSensor_DosingPIT1.getState() = E_DeviceState.OUT_OF_RANGE OR
	fbDosingPump_NutrientA.getState() = E_DeviceState.RUNNING OR
	fbDosingPump_NutrientC.getState() = E_DeviceState.RUNNING OR
	fbDosingPump_phUp.getState() = E_DeviceState.RUNNING OR
	fbDosingPump_phDown.getState() = E_DeviceState.RUNNING  THEN
	
		checkStartPermissive_DosingPump_NutrientB := FALSE;

ELSE
		checkStartPermissive_DosingPump_NutrientB := TRUE;
END_IF
END_METHOD

METHOD checkStartPermissive_DosingPump_NutrientC : BOOL
VAR_INPUT
END_VAR

IF fbSensor_DosingPIT1.getState() = E_DeviceState.OUT_OF_RANGE OR
	fbDosingPump_NutrientA.getState() = E_DeviceState.RUNNING OR
	fbDosingPump_NutrientB.getState() = E_DeviceState.RUNNING OR
	fbDosingPump_phUp.getState() = E_DeviceState.RUNNING OR
	fbDosingPump_phDown.getState() = E_DeviceState.RUNNING  THEN
	
		checkStartPermissive_DosingPump_NutrientC := FALSE;

ELSE
		checkStartPermissive_DosingPump_NutrientC := TRUE;
END_IF
END_METHOD

METHOD checkStartPermissive_DosingPump_phDown : BOOL
VAR_INPUT
END_VAR

IF fbSensor_DosingPIT1.getState() = E_DeviceState.OUT_OF_RANGE OR
	fbDosingPump_NutrientA.getState() = E_DeviceState.RUNNING OR
	fbDosingPump_NutrientB.getState() = E_DeviceState.RUNNING OR
	fbDosingPump_NutrientC.getState() = E_DeviceState.RUNNING OR
	fbDosingPump_phUp.getState() = E_DeviceState.RUNNING  THEN
	
		checkStartPermissive_DosingPump_phDown := FALSE;

ELSE
		checkStartPermissive_DosingPump_phDown := TRUE;
END_IF
END_METHOD

METHOD checkStartPermissive_DosingPump_phUp : BOOL
VAR_INPUT
END_VAR

IF fbSensor_DosingPIT1.getState() = E_DeviceState.OUT_OF_RANGE OR
	fbDosingPump_NutrientA.getState() = E_DeviceState.RUNNING OR
	fbDosingPump_NutrientB.getState() = E_DeviceState.RUNNING OR
	fbDosingPump_NutrientC.getState() = E_DeviceState.RUNNING OR
	fbDosingPump_phDown.getState() = E_DeviceState.RUNNING  THEN
	
		checkStartPermissive_DosingPump_phUp := FALSE;

ELSE
		checkStartPermissive_DosingPump_phUp := TRUE;
END_IF
END_METHOD

METHOD checkStartPermissive_OxyInjector : BOOL
VAR_INPUT
END_VAR

IF fbSumpDosing.getState() = E_DeviceState.OUT_OF_RANGE THEN

		checkStartPermissive_OxyInjector := FALSE;
ELSE
		checkStartPermissive_OxyInjector := TRUE;
END_IF
END_METHOD

METHOD checkStartPermissive_PumpMainPumpA : BOOL
VAR_INPUT
END_VAR

IF fbPump_MainPumpB.getState() = E_DeviceState.RUNNING OR
	(fbValve_IrrigatorSupply.getState() = E_DeviceState.CLOSED AND
		fbValve_WasteWaterReturn.getState() = E_DeviceState.CLOSED AND
		fbSensor_DosingPIT1.getState() = E_DeviceState.LOW_LOW) OR
	fbSumpDosing.getState() = E_DeviceState.LOW_LOW OR
	fbBagFilter1.getDiffPressure() > nPressureDiffLimit_Filter1_Limit OR
	fbBagFilter2.getDiffPressure() > nPressureDiffLimit_Filter2_Limit THEN
	
		checkStartPermissive_PumpMainPumpA := FALSE;
ELSE
	checkStartPermissive_PumpMainPumpA := TRUE;
END_IF
END_METHOD

METHOD checkStartPermissive_PumpMainPumpB : BOOL
VAR_INPUT
END_VAR

IF fbPump_MainPumpA.getState() = E_DeviceState.RUNNING OR
	(fbValve_IrrigatorSupply.getState() = E_DeviceState.CLOSED AND
		fbValve_WasteWaterReturn.getState() = E_DeviceState.CLOSED AND
		fbSensor_DosingPIT1.getState() = E_DeviceState.LOW_LOW) OR
	fbSumpDosing.getState() = E_DeviceState.LOW_LOW OR
	fbBagFilter1.getDiffPressure() > nPressureDiffLimit_Filter1_Limit OR
	fbBagFilter2.getDiffPressure() > nPressureDiffLimit_Filter2_Limit THEN
	
		checkStartPermissive_PumpMainPumpB := FALSE;
ELSE
	checkStartPermissive_PumpMainPumpB := TRUE;
END_IF
END_METHOD

METHOD checkStartPermissive_UltraSonCleaner : BOOL
VAR_INPUT
END_VAR

IF fbSumpDosing.getState() = E_DeviceState.LOW_LOW THEN
	
	checkStartPermissive_UltraSonCleaner := TRUE;
ELSE
	checkStartPermissive_UltraSonCleaner := FALSE;
END_IF
END_METHOD

METHOD checkStartPermissive_UVFilter : BOOL
VAR_INPUT
END_VAR

IF fbSumpDosing.getState() = E_DeviceState.LOW_LOW THEN
	
	checkStartPermissive_UVFilter := FALSE;
ELSE
	checkStartPermissive_UVFilter := TRUE;
END_IF
END_METHOD

METHOD checkStartPermissive_ValveIrrigatorSupply : BOOL
VAR_INPUT
END_VAR
IF  checkWaterQuality() = FALSE THEN
	checkStartPermissive_ValveIrrigatorSupply := FALSE;
ELSE
	checkStartPermissive_ValveIrrigatorSupply := TRUE;
END_IF
END_METHOD

METHOD checkStartPermissive_ValveWasteWaterReturn : BOOL
VAR_INPUT
END_VAR

IF FALSE THEN
	checkStartPermissive_ValveWasteWaterReturn := TRUE;
ELSE
	checkStartPermissive_ValveWasteWaterReturn := FALSE;
END_IF
END_METHOD

METHOD checkWaterQuality : BOOL
VAR_INPUT
END_VAR
checkWaterQuality := TRUE;

IF fbSensor_DissOx.getValue() < nDO_Low_Limit OR
	fbSensor_DissOx.getValue() > nDO_High_Limit THEN
	
	checkWaterQuality := FALSE;
	// raise an event
END_IF

IF fbSensor_EC.getValue() < nEC_Low_Limit OR
	fbSensor_EC.getValue() > nEC_High_Limit THEN
	
	checkWaterQuality := FALSE;
	// raise an event
END_IF


IF fbSensor_ORP.getValue() < nORP_Low_Limit OR
	fbSensor_ORP.getValue() > nORP_High_Limit THEN
	
	checkWaterQuality := FALSE;
	// raise an event
END_IF


IF fbSensor_PH.getValue() < nPH_Low_Limit OR
	fbSensor_PH.getValue() > nPH_High_Limit THEN
	
	checkWaterQuality := FALSE;
	// raise an event
END_IF


IF fbSensor_TMP.getValue() < nTemp_Low_Limit OR
	fbSensor_TMP.getValue() > nTemp_High_Limit THEN
	
	checkWaterQuality := FALSE;
	// raise an event
END_IF
END_METHOD

METHOD devices_init : BOOL
VAR_INPUT
END_VAR
stAllComponents.fbTank_pHUP :=  fbTank_pHUP;
stAllComponents.fbTank_pHDown :=  fbTank_pHDown;
stAllComponents.fbTank_NutrientA :=  fbTank_NutrientA;
stAllComponents.fbTank_NutrientB :=  fbTank_NutrientB;
stAllComponents.fbTank_NutrientC :=  fbTank_NutrientC;

stAllComponents.fbDosingPump_phUp  :=  fbDosingPump_phUp ;
stAllComponents.fbDosingPump_phDown  :=  fbDosingPump_phDown ;


stAllComponents.fbSensor_DissOx1 :=  fbSensor_DissOx1;
stAllComponents.fbSensor_DissOx2 :=  fbSensor_DissOx2;
stAllComponents.fbSensor_EC1 :=  fbSensor_EC1;
stAllComponents.fbSensor_EC2 :=  fbSensor_EC2;
stAllComponents.fbSensor_ORP1 :=  fbSensor_ORP1;
stAllComponents.fbSensor_ORP2 :=  fbSensor_ORP2;
stAllComponents.fbSensor_PH1 :=  fbSensor_PH1;
stAllComponents.fbSensor_PH2 :=  fbSensor_PH2;

stAllComponents.fbSensor_TMP1 :=  fbSensor_TMP1;
stAllComponents.fbSensor_TMP2 :=  fbSensor_TMP2;
stAllComponents.fbSensor_SumpLIT1 :=  fbSensor_SumpLIT1;
stAllComponents.fbSensor_FilterPIT1 :=  fbSensor_FilterPIT1;
stAllComponents.fbSensor_FilterPIT2 :=  fbSensor_FilterPIT2;
stAllComponents.fbSensor_FilterPIT3 :=  fbSensor_FilterPIT3;
stAllComponents.fbSensor_DosingPIT1 :=  fbSensor_DosingPIT1;


stAllComponents.fbValve_DosingSupply := fbValve_DosingSupply;
stAllComponents.fbValve_IrrigatorSupply :=  fbValve_IrrigatorSupply;
stAllComponents.fbValve_WasteWaterReturn :=  fbValve_WasteWaterReturn;


stAllComponents.fbUnit_OxyInjector :=  fbUnit_OxyInjector;
stAllComponents.fbUnit_UltraSonCleaner :=  fbUnit_UltraSonCleaner;


stAllComponents.fbPump_MainPumpA :=  fbPump_MainPumpA;
stAllComponents.fbPump_MainPumpB :=  fbPump_MainPumpB;
stAllComponents.fbDrumFilter1 :=  fbDrumFilter1;
stAllComponents.fbUVFilter1 :=  fbUVFilter1;


stAllComponents.fbBagFilter1 :=  fbBagFilter1;
stAllComponents.fbBagFilter2 :=  fbBagFilter2;
stAllComponents.fbSumpDosing :=  fbSumpDosing;
END_METHOD

METHOD FB_init : BOOL
VAR_INPUT
	bInitRetains : BOOL; // if TRUE, the retain variables are initialized (warm start / cold start)
	bInCopyCode : BOOL;  // if TRUE, the instance afterwards gets moved into the copy code (online change)
	
	
	ModbusMaster: FB_ModbusMaster;
	
	Tank_PHUp: FB_Tank(	TankID:= '', TankDescr:= '');
	Tank_PHDown: FB_Tank(	TankID:= '', TankDescr:= '');
	Tank_NutrientA: FB_Tank(	TankID:= '', TankDescr:= '');
	Tank_NutrientB: FB_Tank(	TankID:= '', TankDescr:= '');
	Tank_NutrientC: FB_Tank(	TankID:= '', TankDescr:= '');
	
	
END_VAR
fbModbusMaster REF= ModbusMaster;


fbTank_pHUP REF= Tank_PHUp;
fbTank_pHDown REF= Tank_pHDown;
fbTank_NutrientA REF= Tank_NutrientA;
fbTank_NutrientB REF= Tank_NutrientB;
fbTank_NutrientC REF= Tank_NutrientC;


(*
fbSequenceManager.addSequence(Sequence := fbSeqDMCal);
fbSequenceManager.addSequence(Sequence := fbSeqDMDrain);
fbSequenceManager.addSequence(Sequence := fbSeqDMFill);
fbSequenceManager.addSequence(Sequence := fbSeqDMMain);

populateComponents();
*)


// populateComponents();
END_METHOD

METHOD setDosingTanks : BOOL
VAR_INPUT
	Tank_pHUP: REFERENCE TO FB_Tank;
	Tank_pHDown: REFERENCE TO FB_Tank;
	Tank_NutrientA: REFERENCE TO FB_Tank;
	Tank_NutrientB: REFERENCE TO FB_Tank;
	Tank_NutrientC: REFERENCE TO FB_Tank;
END_VAR
fbTank_pHUP := Tank_pHUP;
fbTank_pHDown := Tank_pHDown;
fbTank_NutrientA := Tank_NutrientA;
fbTank_NutrientB := Tank_NutrientB;
fbTank_NutrientC := Tank_NutrientC;
END_METHOD

END_FUNCTION_BLOCK

// ---- POUs/06 Machines/_ss/FB_Machine_RND_DosingMachine.TcPOU
{attribute 'OPC.UA.DA.StructuredType' := '1'}
FUNCTION_BLOCK FB_Machine_RND_DosingMachine EXTENDS FB_BaseMachine IMPLEMENTS I_Machine



VAR_IN_OUT
	// Hold a reference to MBMaster - may need to share this with other dosing machines if only 1 x RS485 card is used for both
	{attribute 'OPC.UA.DA' := '0'}
	fbModbusMaster: 	FB_ModbusMaster;                
	
	{attribute 'OPC.UA.DA' := '0'}
	nAgrowtekModbusID: INT;
	
	stInputs: ST_INPUTS_RND_DosingMachine;
END_VAR



VAR
	{attribute 'OPC.UA.DA' := '0'}
	bIsFirstRun: BOOL := TRUE;
	
	//  MACHINE SPECIFIC INPUTS AND OUTPUTS
	// Dosing / Nutrient Limits & SetPoints
	{attribute 'OPC.UA.DA' := '1'}
	nEC_Low_Limit: REAL := 1000;
	{attribute 'OPC.UA.DA' := '1'}
	nEC_High_Limit: REAL := 1400;
	{attribute 'OPC.UA.DA' := '1'}
	nEC_SetPoint: REAL := 1200;
	
	{attribute 'OPC.UA.DA' := '1'}
	nPH_Low_Limit: REAL := 7.8;
	{attribute 'OPC.UA.DA' := '1'}
	nPH_High_Limit: REAL := 8.0;
	{attribute 'OPC.UA.DA' := '1'}
	nPH_SetPoint: REAL := 8.2;
	
	{attribute 'OPC.UA.DA' := '1'}
	nDO_Low_Limit: REAL := 500;
	{attribute 'OPC.UA.DA' := '1'}
	nDO_High_Limit: REAL := 700;
	{attribute 'OPC.UA.DA' := '1'}
	nDO_SetPoint: REAL := 600;
	
	{attribute 'OPC.UA.DA' := '1'}
	nORP_Low_Limit: REAL := 1000;
	{attribute 'OPC.UA.DA' := '1'}
	nORP_High_Limit: REAL := 1200;
	{attribute 'OPC.UA.DA' := '1'}
	nORP_SetPoint: REAL := 1400;
	
	{attribute 'OPC.UA.DA' := '1'}
	nTemp_Low_Limit: REAL  := 1.5;
	{attribute 'OPC.UA.DA' := '1'}
	nTemp_High_Limit: REAL := 26;
	{attribute 'OPC.UA.DA' := '1'}
	nTemp_SetPoint: REAL := 18;  // not applicable ... yet?
	
	// Pressure Setpoints
	{attribute 'OPC.UA.DA' := '1'}
	nPressureMin_Dosing: UINT := 200; //kPA
	{attribute 'OPC.UA.DA' := '1'}
	nPressureMax_Dosing: UINT := 1000; // kPA
	{attribute 'OPC.UA.DA' := '1'}
	nBagFilterPressureMax: UINT := 2000; //kPA
	
	
	// Machine State Flags
	{attribute 'OPC.UA.DA' := '1'}
	bCalibrate_PH: BOOL;
	{attribute 'OPC.UA.DA' := '1'}
	bCalibrate_EC: BOOL;
	{attribute 'OPC.UA.DA' := '1'}
	bCalibrate_ORP: BOOL;
	{attribute 'OPC.UA.DA' := '1'}
	bCalibrate_TEMP: BOOL;
	{attribute 'OPC.UA.DA' := '1'}
	bCalibrate_DO: BOOL;
	{attribute 'OPC.UA.DA' := '1'}
	bCalibrationInProgress: BOOL;	// Used for circulation pump interlock

	
	// Sensors
	{attribute 'OPC.UA.DA' := '1'}
  	{attribute 'OPC.UA.DA.StructuredType' := '1'}
	fbSensor_DissOx: 			FB_Sensor_AtlasDO(SensorID:= 'DO1' , SensorDescr:= ' Dissolved Oxygen - Sensor 1', SensorType:= E_SensorType.Analogue);
	{attribute 'OPC.UA.DA' := '1'}
  	{attribute 'OPC.UA.DA.StructuredType' := '1'}
	fbSensor_EC: 				FB_Sensor_AtlasEC(SensorID:= 'EC1', SensorDescr:= ' Electrical Conductivity - Sensor 1', SensorType:= E_SensorType.Analogue);
	{attribute 'OPC.UA.DA' := '1'}
  	{attribute 'OPC.UA.DA.StructuredType' := '1'}
	fbSensor_ORP: 				FB_Sensor_AtlasORP(SensorID:= 'ORP1', SensorDescr:= ' Oxidation / Reduction Potential - Sensor 1', SensorType:= E_SensorType.Analogue);
	{attribute 'OPC.UA.DA' := '1'}
  	{attribute 'OPC.UA.DA.StructuredType' := '1'}
	fbSensor_PH: 				FB_Sensor_AtlasPH(SensorID:= 'PH1', SensorDescr:= ' Potential Hydrogen (ph) - Sensor 1', SensorType:= E_SensorType.Analogue);
	{attribute 'OPC.UA.DA' := '1'}
  	{attribute 'OPC.UA.DA.StructuredType' := '1'}
	fbSensor_TMP: 				FB_Sensor_AtlasTEMP(SensorID:= 'TMP1', SensorDescr:= 'Water Temperature - Sensor 1', SensorType:= E_SensorType.Analogue);
	{attribute 'OPC.UA.DA' := '1'}
  	{attribute 'OPC.UA.DA.StructuredType' := '1'}
	fbSensor_SumpLSH :  		FB_Sensor_SICKLevelSwitch_GRF18S(SensorID:= 'TK1-LS1', SensorDescr:= '200L Holding Tank Level High', SensorType:= E_SensorType.Analogue);
	{attribute 'OPC.UA.DA' := '1'}
  	{attribute 'OPC.UA.DA.StructuredType' := '1'} 
	fbSensor_FilterPIT1: 		FB_Sensor_OceanControlsPressureTx_BVS006NA( SensorID:= 'PIT1',	SensorDescr:= 'Irrigation Supply Pressure Transmitter 1', SensorType:= E_SensorType.Analogue);
	{attribute 'OPC.UA.DA' := '1'}
  	{attribute 'OPC.UA.DA.StructuredType' := '1'}
	fbSensor_FilterPIT2: 		FB_Sensor_OceanControlsPressureTx_BVS006NA( SensorID:= 'PIT2',	SensorDescr:= 'Irrigation Supply Pressure Transmitter 2', SensorType:= E_SensorType.Analogue);
	{attribute 'OPC.UA.DA' := '1'}
  	{attribute 'OPC.UA.DA.StructuredType' := '1'}  
	fbSensor_DosingPIT1: 		FB_Sensor_OceanControlsPressureTx_BVS006NA( SensorID:= 'PIT3',	SensorDescr:= 'Dosing Line Pressure Transmitter', SensorType:= E_SensorType.Analogue);
	
	
	
	
	
	// Actuators
	{attribute 'OPC.UA.DA' := '1'}
  	{attribute 'OPC.UA.DA.StructuredType' := '1'}
	fbDosingPump_phUp		: FB_DosingPumpAgrowtek(PumpID := 'DP1', PumpDescription := 'Dosing Pump - pH Up', PumpType := E_DosingPump.PH_UP);
	{attribute 'OPC.UA.DA' := '1'}
  	{attribute 'OPC.UA.DA.StructuredType' := '1'}
	fbDosingPump_phDown		: FB_DosingPumpAgrowtek(PumpID := 'DP2', PumpDescription := 'Dosing Pump - pH Down', PumpType := E_DosingPump.PH_DOWN);
	{attribute 'OPC.UA.DA' := '1'}
  	{attribute 'OPC.UA.DA.StructuredType' := '1'}
	fbDosingPump_NutrientA	: FB_DosingPumpAgrowtek(PumpID := 'DP3', PumpDescription := 'Dosing Pump - Nutrient A', PumpType := E_DosingPump.NUTRIENT_A);
	{attribute 'OPC.UA.DA' := '1'}
  	{attribute 'OPC.UA.DA.StructuredType' := '1'}	
	fbDosingPump_NutrientB	: FB_DosingPumpAgrowtek(PumpID := 'DP4', PumpDescription := 'Dosing Pump - Nutrient B', PumpType := E_DosingPump.NUTRIENT_B);
	{attribute 'OPC.UA.DA' := '1'}
  	{attribute 'OPC.UA.DA.StructuredType' := '1'}
	fbDosingPump_NutrientC	: FB_DosingPumpAgrowtek(PumpID := 'DP5', PumpDescription := 'Dosing Pump - Nutrient C', PumpType := E_DosingPump.NUTRIENT_C);
	
	

	
	{attribute 'OPC.UA.DA' := '1'}
  	{attribute 'OPC.UA.DA.StructuredType' := '1'}
	fbValve_RevOsSupply: 		FB_Valve_ONOFF_woMonitoring(ValveID:= 'V5', ValveDescr:= 'Reverse Osmosis Water Supply Valve' );
	{attribute 'OPC.UA.DA' := '1'}
  	{attribute 'OPC.UA.DA.StructuredType' := '1'} 
	fbValve_IrrigatorSupply: 	FB_Valve_ONOFF_woMonitoring(ValveID:= 'V6', ValveDescr:= 'Irrigator Supply Valve' );
	{attribute 'OPC.UA.DA' := '1'}
  	{attribute 'OPC.UA.DA.StructuredType' := '1'} 
	fbPump_MainPumpA: 		FB_PumpDOL_Onga413_RND(PumpID:='PU1' , PumpDescr:='Circulation Pump');
	{attribute 'OPC.UA.DA' := '1'}
  	{attribute 'OPC.UA.DA.StructuredType' := '1'}	 
	fbUVFilter1: 				FB_UVFilter_Pentair_EU40(UnitID:= 'UVC1', UnitDescr:= 'Ultraviolet Filter' );
	{attribute 'OPC.UA.DA' := '1'}
  	{attribute 'OPC.UA.DA.StructuredType' := '1'}	 
	fbSumpDosing: 				FB_Tank(TankID:= 'TK1', TankDescr:= 'Dosing Tank 200L');  
	
	
	// Vendor Units	
	{attribute 'OPC.UA.DA' := '1'}
  	{attribute 'OPC.UA.DA.StructuredType' := '1'} 
	fbUnit_OxyInjector: 		FB_OxygenInjector(UnitID:= 'OXY1' , UnitDescr:= ' Oxygen Injector');
	
